METHOD INTERNAL GetNumberOfAssertsForTest : UINT
VAR_INPUT
    CompleteTestInstancePath : T_MaxString;
END_VAR
VAR
    Counter : UINT;
    NumberOfAsserts : UINT := 0;
END_VAR
IF TotalAsserts > 0 THEN
    FOR Counter := 1 TO TotalAsserts BY 1 DO
        IF AssertResults[Counter].TestInstancePath = CompleteTestInstancePath THEN
            NumberOfAsserts := NumberOfAsserts + 1;
        END_IF
    END_FOR
END_IF

GetNumberOfAssertsForTest := NumberOfAsserts;
END_METHOD

(*
    This method is called in every assert and returns whether this particular assert has already been called.
    The reason one would like to know whether this assert has already been reported or not is to not report it several
    times to any logging service. Because a test-suite can consist of several tests, and certain tests can require the
    test to run over several cycles it means that certain asserts could be called several times and thus we need to
    keep track of which asserts we've already reported. The user of the framework should not need to care for any of
    this and he/she should be able to call the asserts in any way they find suitable.

    To know what assert this is we need to check for the total combination of:
    - Test message
    - Test instance path
    - Expected value
    - Actual value
    Theoretically we can have a situation where a test has three different asserts, each and one with the same test
    message/test instance path/actual value/expected value but called within the same or different cycles. In order for
    us to handle all situations we need a simple algorithm that works according to:
    - Keep track of how many instances the combination of test message/test instance path/expected value/actual value
      we have. So for example, if we have called Assert(Exp := 5, Act := 5, 'Hello there', 'PRG.InstanceTestSuite.Test')
      two times in one cycle, we have two instances of that combination. This is done according to:
    - Iterate all existing reports.
      - If we have a new PLC-cycle, set the current detection-count to zero.
      - If new report does not match in any of the above fields, create it (together with current PLC-cycle).
        Also store the information that we have one instance of this combination and +1 on the detection-count.
      - If new report matches in all of the above, +1 in the detection-count. If this detection-count is larger than
        the stored detection-count for this combination, create a new report and add +1 to the storage of
        the detection-count.
*)
METHOD INTERNAL ReportResult
VAR_INPUT
    ExpectedSize : UDINT;
    ExpectedTypeClass : IBaseLibrary.TypeClass;
    ExpectedValue : POINTER TO BYTE;
    ActualSize : UDINT;
    ActualTypeClass : IBaseLibrary.TypeClass;
    ActualValue : POINTER TO BYTE;
    Message : T_MaxString;
    TestInstancePath : T_MaxString;
END_VAR
VAR_OUTPUT
    AlreadyReported : BOOL := FALSE;
END_VAR
VAR
    LocationIndex : UINT;
    DataTypesNotEquals : BOOL;
    DataSizeNotEquals : BOOL;
    DataContentNotEquals : BOOL;
    CurrentCycleCount : UDINT;
    IteratorCounter : UINT;
    DetectionCountTemp : UINT := 0;
    FoundOne : BOOL;
    AdditionalIdenticalAssert : BOOL;
END_VAR
IF NOT FirstCycleExecuted THEN
    GetCurrentTaskIndex();
    FirstCycleExecuted := TRUE;
END_IF

CurrentCycleCount := TwinCAT_SystemInfoVarList._TaskInfo[GetCurrentTaskIndex.index].CycleCount;
(* Is current cycle the same as the last call to this method?
   If not, reset the detection count *)
IF CurrentCycleCount <> CycleCount THEN
    CopyDetectionCountAndResetDetectionCountInThisCycle();
END_IF

FOR IteratorCounter := 1 TO TotalAsserts BY 1 DO
      IF F_IsAnyEqualToUnionValue(ExpectedOrActual := AssertResultInstances[IteratorCounter].AssertResult.Expected,
                                  ExpectedOrActualSize := ExpectedSize,
                                  ExpectedOrActualTypeClass := ExpectedTypeClass,
                                  ExpectedOrActualValue := ExpectedValue) AND
         F_IsAnyEqualToUnionValue(ExpectedOrActual := AssertResultInstances[IteratorCounter].AssertResult.Actual,
                                  ExpectedOrActualSize := ActualSize,
                                  ExpectedOrActualTypeClass := ActualTypeClass,
                                  ExpectedOrActualValue := ActualValue) AND
        AssertResultInstances[IteratorCounter].AssertResult.Message = Message AND
        AssertResultInstances[IteratorCounter].AssertResult.TestInstancePath = TestInstancePath THEN
            AssertResultInstances[IteratorCounter].DetectionCountThisCycle :=
                AssertResultInstances[IteratorCounter].DetectionCountThisCycle + 1;
            FoundOne := TRUE;
        IF AssertResultInstances[IteratorCounter].DetectionCountThisCycle >
            AssertResultInstances[IteratorCounter].DetectionCount THEN // This assert is new
            AdditionalIdenticalAssert := TRUE;
        END_IF
        EXIT;
    END_IF
END_FOR

// If not found anything, create the first
IF NOT FoundOne THEN
    // No existing match found, create a new entry
    AddAssertResult(ExpectedSize := ExpectedSize,
                    ExpectedTypeClass := ExpectedTypeClass,
                    ExpectedValue := ExpectedValue,
                    ActualSize := ActualSize,
                    ActualTypeClass := ActualTypeClass,
                    ActualValue := ActualValue,
                    Message := Message, TestInstancePath := TestInstancePath);

    CreateAssertResultInstance(ExpectedSize := ExpectedSize,
                               ExpectedTypeClass := ExpectedTypeClass,
                               ExpectedValue := ExpectedValue,
                               ActualSize := ActualSize,
                               ActualTypeClass := ActualTypeClass,
                               ActualValue := ActualValue,
                               Message := Message, TestInstancePath := TestInstancePath);
// An additional instance of this assert needs to be created
ELSIF AdditionalIdenticalAssert THEN
    AddAssertResult(ExpectedSize := ExpectedSize,
                    ExpectedTypeClass := ExpectedTypeClass,
                    ExpectedValue := ExpectedValue,
                    ActualSize := ActualSize,
                    ActualTypeClass := ActualTypeClass,
                    ActualValue := ActualValue,
                    Message := Message, TestInstancePath := TestInstancePath);
// In all other cases, this assert has already been reported, we don't need to do anything
ELSE
    AlreadyReported := TRUE;
END_IF

// Update the cycle count
CycleCount := TwinCAT_SystemInfoVarList._TaskInfo[GetCurrentTaskIndex.index].CycleCount;
END_METHOD

END_FUNCTION_BLOCK

// POUs/FB_FileControl
// This functionblock can open, close, read, write and delete files on the local filesystem
FUNCTION_BLOCK FB_FileControl
VAR
    FileAccessMode : SysFile.ACCESS_MODE := SysFile.AM_APPEND_PLUS; // Append_Plus creates the file if it doesn't exist yet. 
    FileHandle : SysFile.SysTypes.RTS_IEC_HANDLE;
END_VAR

// Closes the currently opened file.
METHOD PUBLIC Close : SysFile.SysTypes.RTS_IEC_RESULT;
IF FileHandle <> SysFile.SysTypes.RTS_INVALID_HANDLE THEN
    Close := SysFile.SysFileClose(hFile := FileHandle);
ELSE
    Close := SysDir.CmpErrors.Errors.ERR_INVALID_HANDLE;
END_IF
END_METHOD

// Deletes a file specified by name, if it exists.
METHOD PUBLIC Delete : SysFile.SysTypes.RTS_IEC_RESULT;
VAR_INPUT
    // File name can contain an absolute or relative path to the file. Path entries must be separated with a forward slash (/)
    FileName : T_MaxString;
END_VAR
Delete := SysFile.SysFileDelete(szFileName := FileName);
END_METHOD

// Opens a file
METHOD PUBLIC Open : SysFile.SysTypes.RTS_IEC_RESULT;
VAR_INPUT
    FileName : T_MaxString := 'filepath/output.xml';  // File name can contain an absolute or relative path to the file. Path entries must be separated with a Slash (/)
    FileAccessMode : SysFile.ACCESS_MODE := SysFile.ACCESS_MODE.AM_APPEND_PLUS;
END_VAR
FileHandle := SysFile.SysFileOpen(szFile := Filename,
                                  am := FileAccessMode,
                                  pResult := ADR(Open));
END_METHOD

// Reads a file from disk into the buffer
METHOD PUBLIC Read : SysFile.SysTypes.RTS_IEC_RESULT;
VAR_INPUT
    BufferPointer : POINTER TO BYTE; // Call with ADR();
    Size : UDINT; // Call with SIZEOF(); 
END_VAR
VAR_OUTPUT
    FileSize : SysFile.SysTypes.RTS_IEC_SIZE;
END_VAR
IF FileHandle <> SysFile.SysTypes.RTS_INVALID_HANDLE THEN
    FileSize := SysFile.SysFileRead(hFile := FileHandle, 
                                    pbyBuffer := BufferPointer,
                                    ulSize := Size,
                                    pResult := ADR(Read));
ELSE
    Read := SysDir.CmpErrors.Errors.ERR_INVALID_HANDLE;
END_IF
END_METHOD

// Writes the contents of the buffer into a file.
METHOD PUBLIC Write : SysFile.SysTypes.RTS_IEC_RESULT;
VAR_INPUT
    BufferPointer : POINTER TO BYTE; // Call with ADR();
    Size : UDINT; // Call with SIZEOF();
END_VAR
IF FileHandle <> SysFile.SysTypes.RTS_INVALID_HANDLE THEN
    SysFile.SysFileWrite(hFile := FileHandle,
                         pbyBuffer := BufferPointer,
                         ulSize := Size,
                         pResult := ADR(Write));
ELSE
    Write := SysDir.CmpErrors.Errors.ERR_INVALID_HANDLE;
END_IF
END_METHOD

END_FUNCTION_BLOCK

// POUs/FB_StreamBuffer
// This functionblock acts as a stream buffer for use with FB_XmlControl
FUNCTION_BLOCK FB_StreamBuffer 
VAR
    _PointerToStringBuffer : POINTER TO BYTE;
    _BufferSize : UDINT;
    _Length : UDINT;
END_VAR

// Appends a string to the buffer
PROPERTY Append : T_MaxString
SET
VAR
    ByteIn : POINTER TO BYTE;
    ByteBuffer : POINTER TO BYTE;
END_VAR
ByteIn := ADR(Append); 
ByteBuffer := _PointerToStringBuffer + _Length; // set start address

WHILE ByteIn^ <> 0 AND (_Length < _BufferSize ) DO
    ByteBuffer^ := ByteIn^; //Copy the 1st byte
    _Length := _Length + 1; // set new buffer length
    ByteIn := ByteIn + 1; // calculate new start address 
    ByteBuffer := ByteBuffer + 1; // calculate new start address 
END_WHILE;

ByteBuffer := _PointerToStringBuffer + _Length; // String End
ByteBuffer^ := 0; // null terminated string
END_SET
END_PROPERTY

// Read current Buffersize
PROPERTY BufferSize : UDINT
GET
BufferSize := _BufferSize;
END_GET
END_PROPERTY

// Clears the buffer and sets the length to 0
METHOD PUBLIC Clear
VAR
	Count : UDINT;
END_VAR
IF (_PointerToStringBuffer = 0) OR (_BufferSize = 0) THEN
    RETURN;
END_IF

FOR Count := 0 TO (_BufferSize - 1) DO
    _PointerToStringBuffer[Count] := 0;
END_FOR

_Length := 0;
END_METHOD

// Copies a string from the character buffer
METHOD PUBLIC Copy : T_MaxString
VAR_INPUT
    StartPos : UDINT;
    EndPos : UDINT;
END_VAR
VAR_OUTPUT
    CopyLen : UDINT;
    XmlError : E_XmlError;
END_VAR
VAR
    Loop : UDINT;
    PointerToByteToCopy : POINTER TO BYTE;
    PointerToBuffer : POINTER TO BYTE;
    CurPos : UDINT;
END_VAR
Loop := 0;
PointerToByteToCopy := ADR(Copy);
PointerToBuffer := _PointerToStringBuffer + StartPos - 1;

WHILE(Loop < SIZEOF(Copy)) AND (StartPos - 1 + Loop < _Length) AND (StartPos + Loop < EndPos) DO
    PointerToByteToCopy^ := PointerToBuffer^;
    Loop := Loop + 1;
    PointerToByteToCopy := ADR(Copy) + Loop;
    PointerToBuffer := _PointerToStringBuffer + StartPos + Loop -1;
END_WHILE;

IF Loop = SIZEOF(Copy) THEN
    XmlError := E_XmlError.ErrorStringLen;
ELSIF StartPos - 1 + Loop = _Length THEN
    XmlError := E_XmlError.ErrorMaxBufferLen;
ELSE
    XmlError := E_XmlError.OK;
END_IF;

PointerToByteToCopy^ := 0;
CopyLen :=  Loop;
END_METHOD

METHOD PUBLIC CutOff : T_MaxString
VAR_INPUT
    StartPos : UDINT;
END_VAR
VAR_OUTPUT
    CutLen : UDINT; 
    XmlError : E_XmlError;
END_VAR
VAR
    Loop : UDINT;
    PointerToByteToCut : POINTER TO BYTE;
    PointerToByteBuffer : POINTER TO BYTE;
END_VAR
Loop := 0;
PointerToByteToCut := ADR(CutOff);
PointerToByteBuffer := _PointerToStringBuffer + StartPos - 1;

WHILE PointerToByteBuffer^ <> 0 AND(Loop < SIZEOF(CutOff)) AND StartPos -1  + Loop < _Length DO
    PointerToByteToCut^ := PointerToByteBuffer^;
    Loop := Loop + 1;
    PointerToByteToCut := ADR(CutOff) + Loop;
    PointerToByteBuffer := _PointerToStringBuffer + StartPos - 1 + Loop;
END_WHILE;

IF PointerToByteBuffer^ = 0 THEN
    XmlError := E_XmlError.OK;
ELSIF Loop = SIZEOF(CutOff) THEN
    XmlError := E_XmlError.ErrorStringLen;
ELSIF StartPos - 1 + Loop = _Length THEN
    XmlError := E_XmlError.ErrorMaxBufferLen;
END_IF;

PointerToByteToCut^ := 0;
_Length := StartPos -1;

PointerToByteBuffer := _PointerToStringBuffer + StartPos - 1;
PointerToByteBuffer^ := 0;

CutLen := Loop;
END_METHOD

(* 
    Find a searchstring in the buffer and returns its position.
    It's possible to add a preffered startposition within buffer
*)
METHOD PUBLIC Find : UDINT
VAR_INPUT
    SearchString : STRING;
    StartPos : UDINT;
END_VAR
VAR
    Loop : UDINT;
    Search : UDINT;
    PointerToBuffer : POINTER TO BYTE;
    PointerToSearch : POINTER TO BYTE;
END_VAR
Loop := 0;
Search := 0;

PointerToBuffer := _PointerToStringBuffer + StartPos;
PointerToSearch := ADR(SearchString);

WHILE(PointerToSearch^ <> 0 ) AND Loop + StartPos < _Length DO
    IF PointerToBuffer^ <> PointerToSearch^ THEN
        Loop := Loop + 1;
        PointerToBuffer := _PointerToStringBuffer + StartPos + Loop;
        PointerToSearch := ADR(SearchString);
        Search := 0;
    ELSE
        Search := Search + 1;
        PointerToBuffer := _PointerToStringBuffer + StartPos + Loop + Search;
        PointerToSearch := ADR(SearchString ) + Search;
    END_IF;
END_WHILE;
Find := Loop + 1 + StartPos;
END_METHOD

METHOD PUBLIC FindBack : UDINT
VAR_INPUT
    SearchString : T_MaxString;
END_VAR
VAR
    Loop : UDINT;
    Search : UDINT;
    PointerToBuffer : POINTER TO BYTE;
    PointerToSearch : POINTER TO BYTE;
END_VAR
Loop := 0;
Search := 0;

PointerToBuffer := _PointerToStringBuffer + _Length;
PointerToSearch := ADR(SearchString);

WHILE(PointerToSearch^ <> 0) AND Loop < _Length DO
    IF PointerToBuffer^ <> PointerToSearch^ THEN
        Loop := Loop + 1;
        PointerToBuffer := _PointerToStringBuffer + _Length - Loop;
        PointerToSearch := ADR(SearchString);
        Search := 0;
    ELSE
        Search := Search + 1;
        PointerToBuffer := _PointerToStringBuffer + _Length - Loop + Search;
        PointerToSearch := ADR(SearchString ) + Search;
    END_IF;
END_WHILE;
FindBack := _Length - Loop + 1;
END_METHOD

// Gets/Sets the current length (in bytes) of the streambuffer
PROPERTY Length : UDINT
GET
Length := _Length;
END_GET
SET
_Length := Length;
END_SET
END_PROPERTY

METHOD PUBLIC SetBuffer : BOOL;
VAR_INPUT
    PointerToBufferAddress : POINTER TO BYTE; // Set buffer address (ADR ...)
    SizeOfBuffer : UDINT; // Set buffer size (SIZEOF ...)
END_VAR
IF (PointerToBufferAddress = 0) OR (SizeOfBuffer = 0) THEN
    SetBuffer := FALSE;
    RETURN;
END_IF;

_BufferSize := SizeOfBuffer;
_PointerToStringBuffer := PointerToBufferAddress;

SetBuffer := TRUE;
END_METHOD

END_FUNCTION_BLOCK

// POUs/FB_XmlControl
(*
    Organizes parsing and composing of XML data. Data can be treated as STRING or char array.
    Buffer size of file can be set via GVL_Param_TcUnit (xUnitBufferSize)
*)
FUNCTION_BLOCK FB_XmlControl
VAR
    XmlBuffer : FB_StreamBuffer;
    TagListBuffer : FB_StreamBuffer;
    Tags : T_MaxString;
    TagListSeekBuffer : FB_StreamBuffer;
    TagsSeek : STRING;
    TagBuffer : FB_StreamBuffer;
    Tag : T_MaxString;
    TagOpen: BOOL;
    Select : UDINT;
    SearchPosition : UDINT; 
END_VAR
VAR CONSTANT
    TAG_OPEN : STRING(1) := '<';
    TAG_CLOSE : STRING(1) := '>';
    END_TAG_CLOSE : STRING(2) := '/>';
    SPACE : STRING(1) := ' ';
    EQUALS : STRING(1) := '=';
    QUOTE : STRING(1) := '"';
    BACK_SLASH : STRING(1) := '\';
    FORWARD_SLASH : STRING(1) := '/';
    OPEN_COMMENT : STRING(5) := '<!-- ';
    CLOSE_COMMENT : STRING(4) := ' -->';
    TAB : STRING(2) := '$T';
    CR_LF : STRING(4) := '$R$N';

    // $OD : ASCII code for carriage return (CR)
    // $$ : to add a $R
    // $' : to add ' (apostrophe)
    // $L or $l : line feed
    // $N or $n : new line
    // $P or $p : next page
    // $R or $r : end of line
END_VAR

// Clears the contents of the entire buffer.
METHOD PUBLIC ClearBuffer
SearchPosition := 0;
TagListSeekBuffer.Length := 0;
XmlBuffer.Length := 0;
TagsSeek := '';
Tag := '';
END_METHOD

(*
    Closes a Tag:
    XML: <MyTag />'

    Method: XML.CloseTag();
*)
METHOD PUBLIC CloseTag : T_MaxString
VAR
    ClosedTag : T_MaxString;
END_VAR
IF TagOpen THEN
    XmlBuffer.Append := END_TAG_CLOSE;
    Select := TagListBuffer.FindBack(SearchString := FORWARD_SLASH);
    ClosedTag := TagListBuffer.CutOff(StartPos := Select);
    TagOpen := FALSE;
ELSE
    Select := TagListBuffer.FindBack(SearchString := FORWARD_SLASH);
    ClosedTag := TagListBuffer.CutOff(StartPos := Select);
    XmlBuffer.Append := TAG_OPEN;
    XmlBuffer.Append := ClosedTag;
    XmlBuffer.Append := TAG_CLOSE;
END_IF

CloseTag := ClosedTag;
END_METHOD

PROPERTY Length : UDINT
GET
Length := XmlBuffer.Length;
END_GET
END_PROPERTY

(*
    Adds a comment
    XML: <!-- MyComment -->

    XML.NewComment(Comment: = 'MyComment');
*)
METHOD PUBLIC NewComment
VAR_INPUT
    Comment : T_MaxString;
END_VAR
IF TagOpen THEN
    XmlBuffer.Append := TAG_CLOSE;
    TagOpen := FALSE;
END_IF;
XmlBuffer.Append := OPEN_COMMENT;
XmlBuffer.Append := Comment;
XmlBuffer.Append := CLOSE_COMMENT;
END_METHOD

(*
    Must be called after opening a new tag

    XML.NewParameter(Name: = 'ParaName', Value: = 'Value');
*)
METHOD PUBLIC NewParameter
VAR_INPUT
    Name : T_MaxString;
    Value : T_MaxString;
END_VAR
XmlBuffer.Append := SPACE;
XmlBuffer.Append := Name;
XmlBuffer.Append := EQUALS;
XmlBuffer.Append := QUOTE;
XmlBuffer.Append := Value;
XmlBuffer.Append := QUOTE;
END_METHOD

(*
    Creates a new Tag:
    XML: <MyTag>

    XML.NewTag(Name: = 'MyTag');
*)
METHOD PUBLIC NewTag
VAR_INPUT
    Name : T_MaxString;
END_VAR
IF TagOpen THEN
    XmlBuffer.Append := TAG_CLOSE;
END_IF;
XmlBuffer.Append := TAG_OPEN;
XmlBuffer.Append := Name;
TagOpen := TRUE;
TagListBuffer.Append := FORWARD_SLASH;
TagListBuffer.Append := Name;
END_METHOD

METHOD PUBLIC NewTagData
VAR_INPUT
    Data : T_MaxString;
END_VAR
XmlBuffer.Append := TAG_CLOSE;
XmlBuffer.Append := Data;
TagOpen := FALSE;
END_METHOD

METHOD PUBLIC SetBuffer
VAR_INPUT
    PointerToBuffer : POINTER TO BYTE; // ADR(..)
    SizeOfBuffer : UDINT; // SIZEOF(..)
END_VAR
XmlBuffer.SetBuffer(PointerToBufferAddress:= PointerToBuffer, SizeOfBuffer := SizeOfBuffer);
TagListBuffer.SetBuffer(PointerToBufferAddress := ADR(Tags), SizeOfBuffer := SIZEOF(Tags));
TagListSeekBuffer.SetBuffer(PointerToBufferAddress := ADR(TagsSeek), SizeOfBuffer := SIZEOF(TagsSeek));
TagBuffer.SetBuffer(PointerToBufferAddress := ADR(Tag), SizeOfBuffer := SIZEOF(Tag));
END_METHOD

(*
    Jump to the beginning of the XML data
    XML.ToStartBuffer();
*)
METHOD PUBLIC ToStartBuffer
SearchPosition := 0;
TagListSeekBuffer.Length := 0;
TagsSeek := '';
Tag := '';
END_METHOD

(*
    Add your own preffered fileheader like:
    XML: <?xml version="1.0" encoding="UTF-8"?>
    
    Start with calling this method before appending any other tags!

    XML.WriteDocumentHeader('<?xml version="1.0" encoding="UTF-8"?>');
*)
METHOD PUBLIC WriteDocumentHeader
VAR_INPUT
    Header : T_MaxString;
END_VAR
XmlBuffer.Append := Header;
END_METHOD

END_FUNCTION_BLOCK

// POUs/FB_TcUnitRunner
// This function block is responsible for holding track of the tests and executing them.
FUNCTION_BLOCK FB_TcUnitRunner
VAR
    // Indication of whether all test suites have reported that they are finished
    AllTestSuitesFinished : BOOL := FALSE;
    AllTestSuitesFinishedTrigger : R_TRIG;

    //Test result information
    TestResults : FB_TestResults;

    (* Prints the results to ADS so that Visual Studio can display the results.
       This test result formatter can be replaced with something else than ADS *)
    AdsTestResultLogger : FB_AdsTestResultLogger(TestResults);
    TestResultLogger : I_TestResultLogger := AdsTestResultLogger;

    (* If this flag is set, it means that some external event triggered the
       request to abort running the test suites *)
    AbortRunningTestSuites : BOOL;

    // Publishes a xUnit compatible XML file
    xUnitXmlPublisher : FB_xUnitXmlPublisher(TestResults);
    XmlTestResultPublisher : I_TestResultLogger := xUnitXmlPublisher;
END_VAR

(* This function sets a flag which makes the runner stop running the tests
   in the test suites *)
METHOD INTERNAL AbortRunningTestSuiteTests
AbortRunningTestSuites := TRUE;
END_METHOD

// This runs all the test suites in parallel
METHOD INTERNAL RunTestSuiteTests
VAR
    Counter : UINT := 0;
    BusyPrinting : BOOL;
    (* We need to hold a temporary state of the statistics 
       as we don't consider the tests to be completely finished until all test suites have executed completely.
       The reason we want to do it this way is because a test suite can run over several cycles. Only once all tests
       are finished (which might take many cycles), do we gather correct statistics *)
    NumberOfTestSuitesFinished : UINT := 0;
END_VAR
IF GVL_TcUnit.StartedAt = 0 THEN
    GVL_TcUnit.StartedAt := F_GetCpuCounterAs64bit(GVL_TcUnit.GetCpuCounter);
END_IF

// Run TcUnit test suites
IF NOT AllTestSuitesFinished THEN
    IF GVL_TcUnit.NumberOfInitializedTestSuites = 0 THEN
        AllTestSuitesFinished := TRUE;
    ELSIF GVL_TcUnit.NumberOfInitializedTestSuites > 0 THEN
        FOR Counter := 1 TO GVL_TcUnit.NumberOfInitializedTestSuites BY 1 DO
            IF GVL_TcUnit.TestSuiteAddresses[Counter]^.AreAllTestsFinished() THEN
                NumberOfTestSuitesFinished := NumberOfTestSuitesFinished + 1;
            ELSE
                GVL_TcUnit.CurrentTestSuiteBeingCalled := GVL_TcUnit.TestSuiteAddresses[Counter];
				GVL_TcUnit.CurrentTestSuiteBeingCalled^.SetStartedAtIfNotSet(Timestamp := F_GetCpuCounterAs64bit(GVL_TcUnit.GetCpuCounter));
                GVL_TcUnit.CurrentTestSuiteBeingCalled^();
				// This is not an efficient way to set the duration
				IF GVL_TcUnit.TestSuiteAddresses[Counter]^.AreAllTestsFinished() THEN
					GVL_TcUnit.CurrentTestSuiteBeingCalled^.CalculateDuration(FinishedAt := F_GetCpuCounterAs64bit(GVL_TcUnit.GetCpuCounter));
				END_IF
            END_IF
        END_FOR
        (* Check if some event triggered an abortion of running the tests, in that case abort it now.
           This can be accomplished by setting the result of the test suites run to finished. *)
        IF AbortRunningTestSuites THEN
            NumberOfTestSuitesFinished := GVL_TcUnit.NumberOfInitializedTestSuites;
        END_IF

        IF NumberOfTestSuitesFinished = GVL_TcUnit.NumberOfInitializedTestSuites THEN
            AllTestSuitesFinished := TRUE;
        END_IF
    END_IF
END_IF

// Store test suite results continuously
TestResults();

// Log test suite results continuously
TestResultLogger.LogTestSuiteResults();

// Publish the xUnit Xml file once if enabled
XmlTestResultPublisher.LogTestSuiteResults();

// Run the buffered ADS logger
GVL_TcUnit.AdsMessageQueue();
END_METHOD

// This runs all the test suites in sequence (one after the other)
METHOD INTERNAL RunTestSuiteTestsInSequence
VAR_INPUT
    TimeBetweenTestSuitesExecution : TIME; // Time delay between a test suite is finished and the next test suite starts
END_VAR
VAR
    BusyPrinting : BOOL;
    (* We need to hold a temporary state of the statistics
       as we don't consider the tests to be completely finished until all test suites have executed completely.
       The reason we want to do it this way is because a test suite can run over several cycles. Only once all tests
       are finished (which might take many cycles), do we gather correct statistics *)
    NumberOfTestSuitesFinished : UINT := 0;
END_VAR
VAR_INST
    (* This variable holds which current test suite is being called, as we are running
       each one in a sequence (one by one) *)
     CurrentlyRunningTestSuite : UINT := 1;
     TimerBetweenExecutionOfTestSuites : TOF;
END_VAR
IF GVL_TcUnit.StartedAt = 0 THEN
    GVL_TcUnit.StartedAt := F_GetCpuCounterAs64bit(GVL_TcUnit.GetCpuCounter);
END_IF

TimerBetweenExecutionOfTestSuites(PT := TimeBetweenTestSuitesExecution);
// Run TcUnit test suites
IF NOT AllTestSuitesFinished THEN
    IF GVL_TcUnit.NumberOfInitializedTestSuites = 0 THEN
        AllTestSuitesFinished := TRUE;
    ELSIF GVL_TcUnit.NumberOfInitializedTestSuites > 0 THEN
        IF TimerBetweenExecutionOfTestSuites.Q THEN
            TimerBetweenExecutionOfTestSuites.IN := FALSE;
        END_IF
        IF GVL_TcUnit.TestSuiteAddresses[CurrentlyRunningTestSuite]^.AreAllTestsFinished() THEN
            IF CurrentlyRunningTestSuite <> GVL_TcUnit.NumberOfInitializedTestSuites THEN
                NumberOfTestSuitesFinished := NumberOfTestSuitesFinished + 1;
                CurrentlyRunningTestSuite := CurrentlyRunningTestSuite + 1;
                TimerBetweenExecutionOfTestSuites.IN := TRUE;
				GVL_TcUnit.CurrentTestSuiteBeingCalled^.CalculateDuration(FinishedAt := F_GetCpuCounterAs64bit(GVL_TcUnit.GetCpuCounter));
            END_IF
        ELSIF NOT TimerBetweenExecutionOfTestSuites.Q THEN
            GVL_TcUnit.CurrentTestSuiteBeingCalled := GVL_TcUnit.TestSuiteAddresses[CurrentlyRunningTestSuite];
			GVL_TcUnit.CurrentTestSuiteBeingCalled^.SetStartedAtIfNotSet(Timestamp := F_GetCpuCounterAs64bit(GVL_TcUnit.GetCpuCounter));
            GVL_TcUnit.CurrentTestSuiteBeingCalled^();
			// This is not an efficient way to set the duration
			IF GVL_TcUnit.TestSuiteAddresses[CurrentlyRunningTestSuite]^.AreAllTestsFinished() THEN
				GVL_TcUnit.CurrentTestSuiteBeingCalled^.CalculateDuration(FinishedAt := F_GetCpuCounterAs64bit(GVL_TcUnit.GetCpuCounter));
			END_IF
        END_IF
        (* Check if some event triggered an abortion of running the tests, in that case abort it now.
           This can be accomplished by setting the result of the test suites run to finished. *)
        IF AbortRunningTestSuites THEN
            NumberOfTestSuitesFinished := GVL_TcUnit.NumberOfInitializedTestSuites;
        END_IF
        IF NumberOfTestSuitesFinished = GVL_TcUnit.NumberOfInitializedTestSuites THEN
            AllTestSuitesFinished := TRUE;
        END_IF
    END_IF
END_IF

// Store test suite results continuously
TestResults();

// Log test suite results continuously
TestResultLogger.LogTestSuiteResults();

// Publish the xUnit Xml file once if enabled
XmlTestResultPublisher.LogTestSuiteResults();

// Run the buffered ADS logger
GVL_TcUnit.AdsMessageQueue();
END_METHOD

END_FUNCTION_BLOCK

// POUs/FB_TestResults
// This function block holds results of the complete test run, i.e. results for all test suites
FUNCTION_BLOCK FB_TestResults IMPLEMENTS I_TestResults
VAR
    // Test results
    TestSuiteResults : ST_TestSuiteResults;

    // Misc variables
    StoringTestSuiteResultNumber : UINT(1..GVL_Param_TcUnit.MaxNumberOfTestSuites);
    StoringTestSuiteTrigger : R_TRIG;
    StoredTestSuiteResults : BOOL;
    StoredGeneralTestResults : BOOL;
    NumberOfTestsToAnalyse : UINT(1..GVL_Param_TcUnit.MaxNumberOfTestsForEachTestSuite);
END_VAR
VAR_TEMP
    TestSuiteName : T_MaxString;
    TestName : T_MaxString;

    TestsInTestSuiteCounter : UINT(1..GVL_Param_TcUnit.MaxNumberOfTestsForEachTestSuite);

    TestToBeStored : FB_Test;
    GeneralTestResultsTestSuitesCounter : UINT(1..GVL_Param_TcUnit.MaxNumberOfTestSuites);
END_VAR

// The body of the function block stores the test results
IF StoringTestSuiteResultNumber <= GVL_TcUnit.NumberOfInitializedTestSuites AND NOT StoredTestSuiteResults THEN
	StoringTestSuiteTrigger(CLK := GVL_TcUnit.TestSuiteAddresses[StoringTestSuiteResultNumber]^.AreAllTestsFinished());

    IF StoringTestSuiteTrigger.Q THEN
        // Remove everything except the program name + "." + test suite name
        TestSuiteName := F_RemoveInstancePathAndProjectNameFromTestInstancePath(TestInstancePath := GVL_TcUnit.TestSuiteAddresses[StoringTestSuiteResultNumber]^.GetInstancePath());

        // Store test suite name and ID
        TestSuiteResults.TestSuiteResults[StoringTestSuiteResultNumber].Name := TestSuiteName;
        TestSuiteResults.TestSuiteResults[StoringTestSuiteResultNumber].Identity := StoringTestSuiteResultNumber - 1;

        // Store number of tests in test suite
        TestSuiteResults.TestSuiteResults[StoringTestSuiteResultNumber].NumberOfTests :=
            GVL_TcUnit.TestSuiteAddresses[StoringTestSuiteResultNumber]^.GetNumberOfTests();

        // Store number of failed tests in test suite
        TestSuiteResults.TestSuiteResults[StoringTestSuiteResultNumber].NumberOfFailedTests :=
            GVL_TcUnit.TestSuiteAddresses[StoringTestSuiteResultNumber]^.GetNumberOfFailedTests();

        // Store the duration
        TestSuiteResults.TestSuiteResults[StoringTestSuiteResultNumber].Duration :=
            GVL_TcUnit.TestSuiteAddresses[StoringTestSuiteResultNumber]^.GetDuration();

        // Limit the test analyse to the max array limit of 'Tests[]' in FB_TestSuite
        NumberOfTestsToAnalyse := GVL_TcUnit.TestSuiteAddresses[StoringTestSuiteResultNumber]^.GetNumberOfTestsToAnalyse();

        // Iterate and print all tests in test suite
        FOR TestsInTestSuiteCounter := 1 TO NumberOfTestsToAnalyse BY 1 DO
            TestToBeStored := GVL_TcUnit.TestSuiteAddresses[StoringTestSuiteResultNumber]^.GetTestByPosition(TestsInTestSuiteCounter);
            // Store test name
            TestSuiteResults.TestSuiteResults[StoringTestSuiteResultNumber].TestCaseResults[TestsInTestSuiteCounter].TestName := TestToBeStored.GetName();

            // Store test class name
            TestSuiteResults.TestSuiteResults[StoringTestSuiteResultNumber].TestCaseResults[TestsInTestSuiteCounter].TestClassName :=
                F_RemoveInstancePathAndProjectNameFromTestInstancePath(GVL_TcUnit.TestSuiteAddresses[StoringTestSuiteResultNumber]^.GetInstancePath());

            // Store whether the test has failed
            TestSuiteResults.TestSuiteResults[StoringTestSuiteResultNumber].TestCaseResults[TestsInTestSuiteCounter].TestIsFailed :=
                TestToBeStored.IsFailed();

            // Store whether the test was skipped
            TestSuiteResults.TestSuiteResults[StoringTestSuiteResultNumber].TestCaseResults[TestsInTestSuiteCounter].TestIsSkipped :=
                TestToBeStored.IsSkipped();

            // Store the (first failed) assertion message
            TestSuiteResults.TestSuiteResults[StoringTestSuiteResultNumber].TestCaseResults[TestsInTestSuiteCounter].FailureMessage :=
                TestToBeStored.GetAssertionMessage();

            // Store the (first failed) assertion type
            TestSuiteResults.TestSuiteResults[StoringTestSuiteResultNumber].TestCaseResults[TestsInTestSuiteCounter].FailureType :=
                TestToBeStored.GetAssertionType();

            // Store number of assertions made
            TestSuiteResults.TestSuiteResults[StoringTestSuiteResultNumber].TestCaseResults[TestsInTestSuiteCounter].NumberOfAsserts :=
                TestToBeStored.GetNumberOfAssertions();

            // Store the duration of the test
            TestSuiteResults.TestSuiteResults[StoringTestSuiteResultNumber].TestCaseResults[TestsInTestSuiteCounter].Duration :=
                TestToBeStored.GetDuration();
        END_FOR

        IF StoringTestSuiteResultNumber = GVL_TcUnit.NumberOfInitializedTestSuites THEN
            StoredTestSuiteResults := TRUE;
        ELSE
            StoringTestSuiteResultNumber := StoringTestSuiteResultNumber + 1;
        END_IF
        StoringTestSuiteTrigger(CLK := FALSE); // Reset trigger
    END_IF
END_IF

(* If all test suites have finished running, store the general test results.
   Take care OF the special CASE where no tests have NOT yet been defined *)
IF GVL_TcUnit.NumberOfInitializedTestSuites = 0 AND (NOT StoredGeneralTestResults) THEN
    StoredGeneralTestResults := TRUE;
    StoredTestSuiteResults := TRUE;
ELSIF StoringTestSuiteResultNumber = GVL_TcUnit.NumberOfInitializedTestSuites AND_THEN
    GVL_TcUnit.TestSuiteAddresses[StoringTestSuiteResultNumber]^.AreAllTestsFinished() AND StoredTestSuiteResults AND (NOT StoredGeneralTestResults) THEN
    TestSuiteResults.NumberOfTestSuites := GVL_TcUnit.NumberOfInitializedTestSuites;
	GVL_TcUnit.Duration := LWORD_TO_LREAL(F_GetCpuCounterAs64bit(GVL_TcUnit.GetCpuCounter) - GVL_TcUnit.StartedAt) * GVL_TcUnit.HundredNanosecondToSecond; // Seconds
    TestSuiteResults.Duration := GVL_TcUnit.Duration;
    FOR GeneralTestResultsTestSuitesCounter := 1 TO GVL_TcUnit.NumberOfInitializedTestSuites BY 1 DO
        TestSuiteResults.NumberOfTestCases := TestSuiteResults.NumberOfTestCases + TestSuiteResults.TestSuiteResults[GeneralTestResultsTestSuitesCounter].NumberOfTests;
        TestSuiteResults.NumberOfSuccessfulTestCases := TestSuiteResults.NumberOfSuccessfulTestCases +
                                                        (TestSuiteResults.TestSuiteResults[GeneralTestResultsTestSuitesCounter].NumberOfTests -
                                                         TestSuiteResults.TestSuiteResults[GeneralTestResultsTestSuitesCounter].NumberOfFailedTests);
        TestSuiteResults.NumberOfFailedTestCases := TestSuiteResults.NumberOfFailedTestCases + TestSuiteResults.TestSuiteResults[GeneralTestResultsTestSuitesCounter].NumberOfFailedTests;
    END_FOR
    StoredGeneralTestResults := TRUE;
END_IF

// Returns whether the storing of the test results is finished
METHOD PUBLIC GetAreTestResultsAvailable : BOOL
GetAreTestResultsAvailable := (StoredTestSuiteResults AND StoredGeneralTestResults);
END_METHOD

METHOD PUBLIC GetTestSuiteResults : REFERENCE TO ST_TestSuiteResults;
GetTestSuiteResults REF=TestSuiteResults;
END_METHOD

END_FUNCTION_BLOCK

// POUs/FB_TestSuite
(* This function block is responsible for holding the internal state of the test suite.
   Every test suite can have one or more tests, and every test can do one or more asserts.
   It's also responsible for providing all the assert-methods for asserting different data types.
   Only failed assertions are recorded.
*)
{attribute 'call_after_init'}
{attribute 'reflection'}
FUNCTION_BLOCK FB_TestSuite
VAR
    {attribute 'instance-path'}
    {attribute 'noinit'}
    InstancePath : T_MaxString;

    (* We need to have access to specific information of the current task that this test suite
       is executed in. This is for instance necessary when we need to know whether a test is
       defined already. The definition of a test that is defined already is that we call on it
       with the same name twice in the same cycle *)
    GetCurrentTaskIndex : GETCURTASKINDEX;

    NumberOfTests : UINT(0..GVL_Param_TcUnit.MaxNumberOfTestsForEachTestSuite) := 0;
    Tests : ARRAY[1..GVL_Param_TcUnit.MaxNumberOfTestsForEachTestSuite] OF FB_Test;
    (* Rising trigger of whether we have already notified the user of that the test name pointed to by the current
       position is a duplicate *)
    TestDuplicateNameTrigger : ARRAY[1..GVL_Param_TcUnit.MaxNumberOfTestsForEachTestSuite] OF R_TRIG;
    (* Last cycle count index for a specific test. Used to detect whether this test has already been defined in the
       current test suite *)
    TestCycleCountIndex : ARRAY[1..GVL_Param_TcUnit.MaxNumberOfTestsForEachTestSuite] OF UDINT;

    AssertResults : FB_AssertResultStatic;
    AssertArrayResults : FB_AssertArrayResultStatic;

    (* Prints the failed asserts to ADS so that Visual Studio can display the assert message.
       This assert formatter can be replaced with something else than ADS *)
    AdsAssertMessageFormatter : FB_AdsAssertMessageFormatter;
    AssertMessageFormatter : I_AssertMessageFormatter := AdsAssertMessageFormatter;

    (* Stores the CPU cycle count with 100ns precision. It also is an indication whether this 
       test suite has started running its tests (> 0 means it has started) *)
    StartedAt : LWORD;

    (* Duration it took to run all tests in this testsuite - including the overhead from TcUnit
       in seconds *)
    Duration : LREAL;

    // Number of ordered tests (created by TEST_ORDERED()) that this test suite contains
    NumberOfOrderedTests : UINT(0..GVL_Param_TcUnit.MaxNumberOfTestsForEachTestSuite);
END_VAR

METHOD INTERNAL AddTest : REFERENCE TO FB_Test
VAR_INPUT
    TestName : T_MaxString;
    IsTestOrdered : BOOL;
END_VAR
VAR
    IteratorCounter : UINT;
    ErrorMessage : T_MaxString;
    TestInstancePath : T_MaxString;
    FunctionCallResult : DINT;
    CycleCount : UDINT;
    TestWithThisNameAlreadyExists : BOOL := FALSE;
    LowerCasedTestName : T_MaxString;
    TrimmedTestName : T_MaxString;
    IgnoreCurrentTestCase : BOOL;
    NumberOfTestsToAnalyse : UINT(1..GVL_Param_TcUnit.MaxNumberOfTestsForEachTestSuite);
END_VAR
GVL_TcUnit.IgnoreCurrentTest := FALSE; // Reset the ignore current test flag

TrimmedTestName := F_LTrim(in := TestName);
TrimmedTestName := F_RTrim(in := TrimmedTestName);
LowerCasedTestName := F_ToLCase(in := TrimmedTestName);

// If test should be disabled, make sure to remove the "disabled_"-part of it from the test name
IF FIND(STR1 := LowerCasedTestName, STR2 := 'disabled_') = 1 THEN
    IgnoreCurrentTestCase := TRUE;
    TrimmedTestName := DELETE(STR := TrimmedTestName, LEN := LEN(STR := 'disabled_'), POS := 1);
END_IF

GetCurrentTaskIndex(); // Gets the task index of where this function block instance is being run in

(* Check if the test name already exists. Make sure there are no other tests with the same name already
   added for this test suite *)

CycleCount := TwinCAT_SystemInfoVarList._TaskInfo[GetCurrentTaskIndex.index].CycleCount;

// Limit the test analyse to the max array limit of 'Tests[]'
NumberOfTestsToAnalyse := GetNumberOfTestsToAnalyse();

// Iterate all the test names that up to this point have been added for this test suite
FOR IteratorCounter := 1 TO NumberOfTestsToAnalyse BY 1 DO
    IF Tests[IteratorCounter].GetName() = TrimmedTestName THEN
        TestWithThisNameAlreadyExists := TRUE;
        // Check if a test with this name has already been called in this PLC cycle
        IF TestCycleCountIndex[IteratorCounter] = CycleCount THEN
            GVL_TcUnit.IgnoreCurrentTest := TRUE;
            (* A test with this name already exists for this test suite and has already been called in this cycle.
               Send a message notification, but only if we have not done so already. *)
            TestDuplicateNameTrigger[IteratorCounter](CLK := TRUE);
            IF TestDuplicateNameTrigger[IteratorCounter].Q THEN // Rising edge detected. We have not reported this before
                TestInstancePath := F_RemoveInstancePathAndProjectNameFromTestInstancePath(TestInstancePath :=
                                                                                           GVL_TcUnit.CurrentTestSuiteBeingCalled^.GetInstancePath());
                ErrorMessage := 'Test with name $'%s$' already exists in test suite $'';
                ErrorMessage := CONCAT(STR1 := ErrorMessage, STR2 := TestInstancePath);
                ErrorMessage := CONCAT(STR1 := ErrorMessage, STR2 := '$'');
                GVL_TcUnit.AdsMessageQueue.WriteLog(MsgCtrlMask := ADSLOG_MSGTYPE_ERROR,
                                                    MsgFmtStr := ErrorMessage,
                                                    StrArg := TrimmedTestName);
            END_IF
        END_IF
        TestCycleCountIndex[IteratorCounter] := CycleCount;
    END_IF
END_FOR

IF NOT TestWithThisNameAlreadyExists THEN
    // Test has not been found. Add it.
    Tests[IteratorCounter].SetName(Name := TrimmedTestName);
    NumberOfTests := NumberOfTests + 1;
    TestCycleCountIndex[NumberOfTests] := CycleCount;
    IF IgnoreCurrentTestCase THEN
        Tests[IteratorCounter].SetSkipped();
    END_IF

    // Extra information to be added if test is ordered (called by TEST_ORDERED())
    IF IsTestOrdered THEN
        NumberOfOrderedTests := NumberOfOrderedTests + 1;
        Tests[IteratorCounter].SetTestOrder(OrderNumber := NumberOfOrderedTests);
    END_IF
END_IF

// Check if this test should be disabled
IF IgnoreCurrentTestCase THEN
    GVL_TcUnit.IgnoreCurrentTest := TRUE;
    RETURN;
END_IF

AddTest REF= GetTestByName(TrimmedTestName);
END_METHOD

METHOD INTERNAL AddTestNameToInstancePath : T_MaxString
VAR_INPUT
    TestInstancePath : T_MaxString;
END_VAR
VAR
    CompleteTestInstancePath : T_MaxString;
END_VAR
CompleteTestInstancePath := CONCAT(STR1 := TestInstancePath, STR2 := '@');
AddTestNameToInstancePath := CONCAT(STR1 := CompleteTestInstancePath, STR2 := GVL_TcUnit.CurrentTestNameBeingCalled);
END_METHOD

METHOD PUBLIC AreAllTestsFinished : BOOL
VAR
    Counter : UINT;
    GetCurTaskIndex : GETCURTASKINDEX;
    NumberOfTestsToAnalyse : UINT(1..GVL_Param_TcUnit.MaxNumberOfTestsForEachTestSuite);
END_VAR
AreAllTestsFinished := FALSE;

IF NumberOfTests > 0 THEN
    AreAllTestsFinished := TRUE;
    // Limit the test analyse to the max array limit of 'Tests[]'
    NumberOfTestsToAnalyse := GetNumberOfTestsToAnalyse();
    // A test is considered finished if it is finished running (i.e. set by TEST_FINISHED) or if it is skipped/disabled
    FOR Counter := 1 TO NumberOfTestsToAnalyse BY 1 DO
        AreAllTestsFinished := AreAllTestsFinished AND (Tests[Counter].IsFinished() OR Tests[Counter].IsSkipped());
    END_FOR
END_IF

(* If we have been running at least one cycle and no tests are registered, it means that this testsuite is empty
   and doesn't contain any test cases. In that case, ignore this testsuite. *)
GetCurTaskIndex();
IF NumberOfTests = 0 AND NOT TwinCAT_SystemInfoVarList._TaskInfo[GetCurTaskIndex.index].FirstCycle AND StartedAt > 0 THEN
	AreAllTestsFinished := TRUE;
END_IF
END_METHOD

// Asserts that two LREAL 2D-arrays are equal to within a positive delta. If they are not, an assertion error is created.
METHOD PUBLIC AssertArray2dEquals_LREAL
VAR_IN_OUT
    Expecteds : ARRAY[*,*] OF LREAL; // LREAL 2d array with expected values
    Actuals : ARRAY[*,*] OF LREAL; // LREAL 2d array with actual values
END_VAR
VAR_INPUT
    Delta : LREAL; // The maximum delta between the value of expected and actual for which both numbers are still considered equal, proportional to the expected value in that array cell
    Message : T_MaxString; // The identifying message for the assertion error
END_VAR
VAR
    Equals : BOOL := TRUE;
    SizeEquals : BOOL := TRUE;
    ExpectedString : T_MaxString;
    ActualString : T_MaxString;
    AlreadyReported : BOOL;
    TestInstancePath : T_MaxString;
    DimensionIndex : USINT; // Index when looping through Dimensions
    LowerBoundExpecteds : ARRAY[1..2] OF DINT; // Lower bounds of Expecteds array in each dimension
    UpperBoundExpecteds : ARRAY[1..2] OF DINT; // Upper bounds of Expecteds array in each dimension
    LowerBoundActuals : ARRAY[1..2] OF DINT; // Lower bounds of Actuals array in each dimension
    UpperBoundActuals : ARRAY[1..2] OF DINT; // Upper bounds of Actuals array in each dimension
    SizeOfExpecteds : ARRAY[1..2] OF DINT; // Size of Expecteds array in each dimension
    SizeOfActuals : ARRAY[1..2] OF DINT; // Size of Actuals array in each dimension
    Offset : ARRAY[1..2] OF DINT; // Current Array index offsets from Lower Bound in each dimension
    ExpectedArrayIndex : ARRAY[1..2] OF DINT; // Array of current Expected array indexes when looping through arrays
    ActualArrayIndex : ARRAY[1..2] OF DINT; // Array of current Actual array indexes when looping through arrays
    Expected : LREAL; // Single expected value
    Actual : LREAL; // Single actual value
END_VAR
IF GVL_TcUnit.IgnoreCurrentTest OR GVL_TcUnit.CurrentTestIsFinished THEN
    RETURN;
END_IF

TestInstancePath := AddTestNameToInstancePath(FindTestSuiteInstancePath());

(* UPPER_BOUND and LOWER_BOUND require literals for their second parameter,
   so they can't be called in a dimension-based loop.
   Thus we copy the array dimensions into arrays which accept variable indexes *)
LowerBoundExpecteds[1] := LOWER_BOUND(Expecteds, 1);
UpperBoundExpecteds[1] := UPPER_BOUND(Expecteds, 1);
LowerBoundExpecteds[2] := LOWER_BOUND(Expecteds, 2);
UpperBoundExpecteds[2] := UPPER_BOUND(Expecteds, 2);
LowerBoundActuals[1] := LOWER_BOUND(Actuals, 1);
UpperBoundActuals[1] := UPPER_BOUND(Actuals, 1);
LowerBoundActuals[2] := LOWER_BOUND(Actuals, 2);
UpperBoundActuals[2] := UPPER_BOUND(Actuals, 2);

FOR DimensionIndex := 1 TO 2 DO
    SizeOfExpecteds[DimensionIndex] := ABS(UpperBoundExpecteds[DimensionIndex] - LowerBoundExpecteds[DimensionIndex]) + 1;
    SizeOfActuals[DimensionIndex] := ABS(UpperBoundActuals[DimensionIndex] - LowerBoundActuals[DimensionIndex]) + 1;

    IF SizeOfExpecteds[DimensionIndex] <> SizeOfActuals[DimensionIndex] THEN
        Equals := FALSE;
        SizeEquals := FALSE;
    END_IF
END_FOR

IF SizeEquals THEN
    (* Even though we know that both arrays are equal in size, the two arrays can start at two completely different
       indexes in each dimension, which needs to be taken into account. *)
    FOR Offset[1] := 0 TO SizeOfExpecteds[1] - 1 DO // Iterate Dimension 1
        FOR Offset[2] := 0 TO SizeOfExpecteds[2] - 1 DO // Iterate Dimension 2
            // Update index variables
            FOR DimensionIndex := 1 TO 2 DO
                ExpectedArrayIndex[DimensionIndex] := LowerBoundExpecteds[DimensionIndex] + Offset[DimensionIndex];
                ActualArrayIndex[DimensionIndex] := LowerBoundActuals[DimensionIndex] + Offset[DimensionIndex];
            END_FOR

            // Get array element values
            Expected := Expecteds[ExpectedArrayIndex[1], ExpectedArrayIndex[2]];
            Actual := Actuals[ActualArrayIndex[1], ActualArrayIndex[2]]; 

            IF ABS(Expected - Actual) > Delta THEN
                Equals := FALSE;
                EXIT;
            END_IF
        END_FOR

        // Check for loop bailout
        IF NOT Equals THEN
            EXIT;
        END_IF
    END_FOR
END_IF

AssertArrayResults.ReportResult(ExpectedsSize := DINT_TO_UDINT(SizeOfExpecteds[1] * SizeOfExpecteds[2]),
                                ExpectedsTypeClass := IBaseLibrary.TypeClass.TYPE_LREAL,
                                ActualsSize := DINT_TO_UDINT(SizeOfActuals[1] * SizeOfActuals[2]),
                                ActualsTypeClass := IBaseLibrary.TypeClass.TYPE_LREAL,
                                Message := Message,
                                TestInstancePath := TestInstancePath,
                                AlreadyReported => AlreadyReported);

IF NOT AlreadyReported AND NOT Equals THEN
    SetTestFailed(AssertionType := E_AssertionType.Type_Array2D_LREAL,
                  AssertionMessage := Message);

    IF NOT SizeEquals THEN
        Message := CONCAT(STR1 := Message, STR2 := ', size of arrays not matching.');
        ExpectedString := 'SIZE = [';
        ExpectedString := CONCAT(STR1 := ExpectedString,STR2 := DINT_TO_STRING(LowerBoundExpecteds[1]));
        ExpectedString := CONCAT(STR1 := ExpectedString, STR2 := '..');
        ExpectedString := CONCAT(STR1 := ExpectedString, STR2 := DINT_TO_STRING(UpperBoundExpecteds[1]));
        ExpectedString := CONCAT(STR1 := ExpectedString, STR2 := ',');
        ExpectedString := CONCAT(STR1 := ExpectedString, STR2 := DINT_TO_STRING(LowerBoundExpecteds[2]));
        ExpectedString := CONCAT(STR1 := ExpectedString, STR2 := '..');
        ExpectedString := CONCAT(STR1 := ExpectedString, STR2 := DINT_TO_STRING(UpperBoundExpecteds[2]));
        ExpectedString := CONCAT(STR1 := ExpectedString, STR2 := '] (');
        ExpectedString := CONCAT(STR1 := ExpectedString, STR2 := DINT_TO_STRING(SizeOfExpecteds[1]));
        ExpectedString := CONCAT(STR1 := ExpectedString, STR2 := 'x');
        ExpectedString := CONCAT(STR1 := ExpectedString, STR2 := DINT_TO_STRING(SizeOfExpecteds[2]));
        ExpectedString := CONCAT(STR1 := ExpectedString, STR2 := ')');

        ActualString := 'SIZE = [';
        ActualString := CONCAT(STR1 := ActualString, STR2 := DINT_TO_STRING(LowerBoundActuals[1]));
        ActualString := CONCAT(STR1 := ActualString, STR2 := '..');
        ActualString := CONCAT(STR1 := ActualString, STR2 := DINT_TO_STRING(UpperBoundActuals[1]));
        ActualString := CONCAT(STR1 := ActualString, STR2 := ',');
        ActualString := CONCAT(STR1 := ActualString, STR2 := DINT_TO_STRING(LowerBoundActuals[2]));
        ActualString := CONCAT(STR1 := ActualString, STR2 := '..');
        ActualString := CONCAT(STR1 := ActualString, STR2 := DINT_TO_STRING(UpperBoundActuals[2]));
        ActualString := CONCAT(STR1 := ActualString, STR2 := '] (');
        ActualString := CONCAT(STR1 := ActualString, STR2 := DINT_TO_STRING(SizeOfActuals[1]));
        ActualString := CONCAT(STR1 := ActualString, STR2 := 'x');
        ActualString := CONCAT(STR1 := ActualString, STR2 := DINT_TO_STRING(SizeOfActuals[2]));
        ActualString := CONCAT(STR1 := ActualString, STR2 := ')');
    ELSE
        ExpectedString := 'ARRAY[';
        ExpectedString := CONCAT(STR1 := ExpectedString, STR2 := DINT_TO_STRING(ExpectedArrayIndex[1]));
        ExpectedString := CONCAT(STR1 := ExpectedString, STR2 := ',');
        ExpectedString := CONCAT(STR1 := ExpectedString, STR2 := DINT_TO_STRING(ExpectedArrayIndex[2]));
        ExpectedString := CONCAT(STR1 := ExpectedString, STR2 := '] = ');
        ExpectedString := CONCAT(STR1 := ExpectedString, STR2 := LREAL_TO_STRING(Expected));

        ActualString := 'ARRAY[';
        ActualString := CONCAT(STR1 := ActualString, STR2 := DINT_TO_STRING(ActualArrayIndex[1]));
        ActualString := CONCAT(STR1 := ActualString, STR2 := ',');
        ActualString := CONCAT(STR1 := ActualString, STR2 := DINT_TO_STRING(ActualArrayIndex[2]));
        ActualString := CONCAT(STR1 := ActualString, STR2 := '] = ');
        ActualString := CONCAT(STR1 := ActualString, STR2 := LREAL_TO_STRING(Actual));
    END_IF

    AssertMessageFormatter.LogAssertFailure(Expected := ExpectedString,
                                            Actual := ActualString,
                                            Message := Message,
                                            TestInstancePath := TestInstancePath);
END_IF
END_METHOD

// Asserts that two REAL 2D-arrays are equal to within a positive delta. If they are not, an assertion error is created.
METHOD PUBLIC AssertArray2dEquals_REAL
VAR_IN_OUT
    Expecteds : ARRAY[*,*] OF REAL; // REAL 2d array with expected values
    Actuals : ARRAY[*,*] OF REAL; // REAL 2d array with actual values
END_VAR
VAR_INPUT
    Delta : REAL; // The maximum delta between the value of expected and actual for which both numbers are still considered equal, proportional to the expected value in that array cell
    Message : T_MaxString; // The identifying message for the assertion error
END_VAR
VAR
    Equals : BOOL := TRUE;
    SizeEquals : BOOL := TRUE;
    ExpectedString : T_MaxString;
    ActualString : T_MaxString;
    AlreadyReported : BOOL;
    TestInstancePath : T_MaxString;
    DimensionIndex : USINT; // Index when looping through Dimensions
    LowerBoundExpecteds : ARRAY[1..2] OF DINT; // Lower bounds of Expecteds array in each dimension
    UpperBoundExpecteds : ARRAY[1..2] OF DINT; // Upper bounds of Expecteds array in each dimension
    LowerBoundActuals : ARRAY[1..2] OF DINT; // Lower bounds of Actuals array in each dimension
    UpperBoundActuals : ARRAY[1..2] OF DINT; // Upper bounds of Actuals array in each dimension
    SizeOfExpecteds : ARRAY[1..2] OF DINT; // Size of Expecteds array in each dimension
    SizeOfActuals : ARRAY[1..2] OF DINT; // Size of Actuals array in each dimension
    Offset : ARRAY[1..2] OF DINT; // Current Array index offsets from Lower Bound in each dimension
    ExpectedArrayIndex : ARRAY[1..2] OF DINT; // Array of current Expected array indexes when looping through arrays
    ActualArrayIndex : ARRAY[1..2] OF DINT; // Array of current Actual array indexes when looping through arrays
    Expected : REAL; // Single expected value
    Actual : REAL; // Single actual value
END_VAR
IF GVL_TcUnit.IgnoreCurrentTest OR GVL_TcUnit.CurrentTestIsFinished THEN
    RETURN;
END_IF

TestInstancePath := AddTestNameToInstancePath(FindTestSuiteInstancePath());

(* UPPER_BOUND and LOWER_BOUND require literals for their second parameter, 
   so they can't be called in a dimension-based loop.
   Thus we copy the ARRAY dimensions into arrays which accept variable indexes *)
LowerBoundExpecteds[1] := LOWER_BOUND(Expecteds, 1);
UpperBoundExpecteds[1] := UPPER_BOUND(Expecteds, 1);
LowerBoundExpecteds[2] := LOWER_BOUND(Expecteds, 2);
UpperBoundExpecteds[2] := UPPER_BOUND(Expecteds, 2);
LowerBoundActuals[1] := LOWER_BOUND(Actuals, 1);
UpperBoundActuals[1] := UPPER_BOUND(Actuals, 1);
LowerBoundActuals[2] := LOWER_BOUND(Actuals, 2);
UpperBoundActuals[2] := UPPER_BOUND(Actuals, 2);

FOR DimensionIndex := 1 TO 2 DO
    SizeOfExpecteds[DimensionIndex] := ABS(UpperBoundExpecteds[DimensionIndex] - LowerBoundExpecteds[DimensionIndex]) + 1;
    SizeOfActuals[DimensionIndex] := ABS(UpperBoundActuals[DimensionIndex] - LowerBoundActuals[DimensionIndex]) + 1;

    IF SizeOfExpecteds[DimensionIndex] <> SizeOfActuals[DimensionIndex] THEN
        Equals := FALSE;
        SizeEquals := FALSE;
    END_IF
END_FOR

IF SizeEquals THEN
    (* Even though we know that both arrays are equal in size, the two arrays can start at two completely different
       indexes in each dimension, which needs to be taken into account. *)
    FOR Offset[1] := 0 TO SizeOfExpecteds[1] - 1 DO // Iterate Dimension 1
        FOR Offset[2] := 0 TO SizeOfExpecteds[2] - 1 DO // Iterate Dimension 2
            // Update index variables
            FOR DimensionIndex := 1 TO 2 DO
                ExpectedArrayIndex[DimensionIndex] := LowerBoundExpecteds[DimensionIndex] + Offset[DimensionIndex];
                ActualArrayIndex[DimensionIndex] := LowerBoundActuals[DimensionIndex] + Offset[DimensionIndex];
            END_FOR

            // Get array element values
            Expected := Expecteds[ExpectedArrayIndex[1], ExpectedArrayIndex[2]];
            Actual := Actuals[ActualArrayIndex[1], ActualArrayIndex[2]]; 

            IF ABS(Expected - Actual) > Delta THEN
                Equals := FALSE;
                EXIT;
            END_IF
        END_FOR

        // Check for loop bailout
        IF NOT Equals THEN
            EXIT;
        END_IF
    END_FOR
END_IF

AssertArrayResults.ReportResult(ExpectedsSize := DINT_TO_UDINT(SizeOfExpecteds[1] * SizeOfExpecteds[2]),
                                ExpectedsTypeClass := IBaseLibrary.TypeClass.TYPE_REAL,
                                ActualsSize := DINT_TO_UDINT(SizeOfActuals[1] * SizeOfActuals[2]),
                                ActualsTypeClass := IBaseLibrary.TypeClass.TYPE_REAL,
                                Message := Message,
                                TestInstancePath := TestInstancePath,
                                AlreadyReported => AlreadyReported);

IF NOT AlreadyReported AND NOT Equals THEN
    SetTestFailed(AssertionType := E_AssertionType.Type_Array2D_REAL,
                  AssertionMessage := Message);

    IF NOT SizeEquals THEN
        Message := CONCAT(STR1 := Message, STR2 := ', size of arrays not matching.');
        ExpectedString := 'SIZE = [';
        ExpectedString := CONCAT(STR1 := ExpectedString, STR2 := DINT_TO_STRING(LowerBoundExpecteds[1]));
        ExpectedString := CONCAT(STR1 := ExpectedString, STR2 := '..');
        ExpectedString := CONCAT(STR1 := ExpectedString, STR2 := DINT_TO_STRING(UpperBoundExpecteds[1]));
        ExpectedString := CONCAT(STR1 := ExpectedString, STR2 := ',');
        ExpectedString := CONCAT(STR1 := ExpectedString, STR2 := DINT_TO_STRING(LowerBoundExpecteds[2]));
        ExpectedString := CONCAT(STR1 := ExpectedString, STR2 := '..');
        ExpectedString := CONCAT(STR1 := ExpectedString, STR2 := DINT_TO_STRING(UpperBoundExpecteds[2]));
        ExpectedString := CONCAT(STR1 := ExpectedString, STR2 := '] (');
        ExpectedString := CONCAT(STR1 := ExpectedString, STR2 := DINT_TO_STRING(SizeOfExpecteds[1]));
        ExpectedString := CONCAT(STR1 := ExpectedString, STR2 := 'x');
        ExpectedString := CONCAT(STR1 := ExpectedString, STR2 := DINT_TO_STRING(SizeOfExpecteds[2]));
        ExpectedString := CONCAT(STR1 := ExpectedString, STR2 := ')');

        ActualString := 'SIZE = [';
        ActualString := CONCAT(STR1 := ActualString, STR2 := DINT_TO_STRING(LowerBoundActuals[1]));
        ActualString := CONCAT(STR1 := ActualString, STR2 := '..');
        ActualString := CONCAT(STR1 := ActualString, STR2 := DINT_TO_STRING(UpperBoundActuals[1]));
        ActualString := CONCAT(STR1 := ActualString, STR2 := ',');
        ActualString := CONCAT(STR1 := ActualString, STR2 := DINT_TO_STRING(LowerBoundActuals[2]));
        ActualString := CONCAT(STR1 := ActualString, STR2 := '..');
        ActualString := CONCAT(STR1 := ActualString, STR2 := DINT_TO_STRING(UpperBoundActuals[2]));
        ActualString := CONCAT(STR1 := ActualString, STR2 := '] (');
        ActualString := CONCAT(STR1 := ActualString, STR2 := DINT_TO_STRING(SizeOfActuals[1]));
        ActualString := CONCAT(STR1 := ActualString, STR2 := 'x');
        ActualString := CONCAT(STR1 := ActualString, STR2 := DINT_TO_STRING(SizeOfActuals[2]));
        ActualString := CONCAT(STR1 := ActualString, STR2 := ')');
    ELSE
        ExpectedString := 'ARRAY[';
        ExpectedString := CONCAT(STR1 := ExpectedString, STR2 := DINT_TO_STRING(ExpectedArrayIndex[1]));
        ExpectedString := CONCAT(STR1 := ExpectedString, STR2 := ',');
        ExpectedString := CONCAT(STR1 := ExpectedString, STR2 := DINT_TO_STRING(ExpectedArrayIndex[2]));
        ExpectedString := CONCAT(STR1 := ExpectedString, STR2 := '] = ');
        ExpectedString := CONCAT(STR1 := ExpectedString, STR2 := REAL_TO_STRING(Expected));

        ActualString := 'ARRAY[';
        ActualString := CONCAT(STR1 := ActualString, STR2 := DINT_TO_STRING(ActualArrayIndex[1]));
        ActualString := CONCAT(STR1 := ActualString, STR2 := ',');
        ActualString := CONCAT(STR1 := ActualString, STR2 := DINT_TO_STRING(ActualArrayIndex[2]));
        ActualString := CONCAT(STR1 := ActualString, STR2 := '] = ');
        ActualString := CONCAT(STR1 := ActualString, STR2 := REAL_TO_STRING(Actual));
    END_IF

    AssertMessageFormatter.LogAssertFailure(Expected := ExpectedString,
                                            Actual := ActualString,
                                            Message := Message,
                                            TestInstancePath := TestInstancePath);
END_IF
END_METHOD

// Asserts that two LREAL 3D-arrays are equal to within a positive delta. If they are not, an assertion error is created.
METHOD PUBLIC AssertArray3dEquals_LREAL
VAR_IN_OUT
    Expecteds : ARRAY[*,*,*] OF LREAL; // LREAL 3d array with expected values
    Actuals : ARRAY[*,*,*] OF LREAL; // LREAL 3d array with actual values
END_VAR
VAR_INPUT
    Delta : LREAL; // The maximum delta between the value of expected and actual for which both numbers are still considered equal, proportional to the expected value in that array cell
    Message : T_MaxString; // The identifying message for the assertion error
END_VAR
VAR
    Equals : BOOL := TRUE;
    SizeEquals : BOOL := TRUE;
    ExpectedString : T_MaxString;
    ActualString : T_MaxString;
    AlreadyReported : BOOL;
    TestInstancePath : T_MaxString;
    DimensionIndex : USINT;  // Index when looping through Dimensions
    LowerBoundExpecteds : ARRAY[1..3] OF DINT; // Lower bounds of Expecteds array in each dimension
    UpperBoundExpecteds : ARRAY[1..3] OF DINT; // Upper bounds of Expecteds array in each dimension
    LowerBoundActuals : ARRAY[1..3] OF DINT; // Lower bounds of Actuals array in each dimension
    UpperBoundActuals : ARRAY[1..3] OF DINT; // Upper bounds of Actuals array in each dimension
    SizeOfExpecteds : ARRAY[1..3] OF DINT; // Size of Expecteds array in each dimension
    SizeOfActuals : ARRAY[1..3] OF DINT; // Size of Actuals array in each dimension
    Offset : ARRAY[1..3] OF DINT; // Current Array index offsets from Lower Bound in each dimension
    ExpectedArrayIndex : ARRAY[1..3] OF DINT; // Array of current Expected array indexes when looping through arrays
    ActualArrayIndex : ARRAY[1..3] OF DINT; // Array of current Actual array indexes when looping through arrays
    Expected : LREAL; // Single expected value
    Actual : LREAL; // Single actual value
END_VAR
IF GVL_TcUnit.IgnoreCurrentTest OR GVL_TcUnit.CurrentTestIsFinished THEN
    RETURN;
END_IF

TestInstancePath := AddTestNameToInstancePath(FindTestSuiteInstancePath());

(* UPPER_BOUND and LOWER_BOUND require literals for their second parameter,
   so they can't be called in a dimension-based loop.
   Thus we copy the array dimensions into arrays which accept variable indexes *)
LowerBoundExpecteds[1] := LOWER_BOUND(Expecteds, 1);
UpperBoundExpecteds[1] := UPPER_BOUND(Expecteds, 1);
LowerBoundExpecteds[2] := LOWER_BOUND(Expecteds, 2);
UpperBoundExpecteds[2] := UPPER_BOUND(Expecteds, 2);
LowerBoundExpecteds[3] := LOWER_BOUND(Expecteds, 3);
UpperBoundExpecteds[3] := UPPER_BOUND(Expecteds, 3);
LowerBoundActuals[1] := LOWER_BOUND(Actuals, 1);
UpperBoundActuals[1] := UPPER_BOUND(Actuals, 1);
LowerBoundActuals[2] := LOWER_BOUND(Actuals, 2);
UpperBoundActuals[2] := UPPER_BOUND(Actuals, 2);
LowerBoundActuals[3] := LOWER_BOUND(Actuals, 3);
UpperBoundActuals[3] := UPPER_BOUND(Actuals, 3);

FOR DimensionIndex := 1 TO 3 DO
    SizeOfExpecteds[DimensionIndex] := ABS(UpperBoundExpecteds[DimensionIndex] - LowerBoundExpecteds[DimensionIndex]) + 1;
    SizeOfActuals[DimensionIndex] := ABS(UpperBoundActuals[DimensionIndex] - LowerBoundActuals[DimensionIndex]) + 1;

    IF SizeOfExpecteds[DimensionIndex] <> SizeOfActuals[DimensionIndex] THEN
        Equals := FALSE;
        SizeEquals := FALSE;
    END_IF
END_FOR

IF SizeEquals THEN
    (* Even though we know that both arrays are equal in size, the three arrays can start at three completely different
       indexes in each dimension, which needs to be taken into account. *)
    FOR Offset[1] := 0 TO SizeOfExpecteds[1] - 1 DO // Iterate Dimension 1
        FOR Offset[2] := 0 TO SizeOfExpecteds[2] - 1 DO // Iterate Dimension 2
            FOR Offset[3] := 0 TO SizeOfExpecteds[3] - 1 DO // Iterate Dimension 3
                // Update index variables
                FOR DimensionIndex := 1 TO 3 DO
                    ExpectedArrayIndex[DimensionIndex] := LowerBoundExpecteds[DimensionIndex] + Offset[DimensionIndex];
                    ActualArrayIndex[DimensionIndex] := LowerBoundActuals[DimensionIndex] + Offset[DimensionIndex];
                END_FOR

                // Get array element values
                Expected := Expecteds[ExpectedArrayIndex[1], ExpectedArrayIndex[2], ExpectedArrayIndex[3]];
                Actual := Actuals[ActualArrayIndex[1], ActualArrayIndex[2], ActualArrayIndex[3]]; 

                IF ABS(Expected - Actual) > Delta THEN
                    Equals := FALSE;
                    EXIT;
                END_IF
            END_FOR

            // Check for loop bailout
            IF NOT Equals THEN
                EXIT;
            END_IF
        END_FOR

        // Check for loop bailout
        IF NOT Equals THEN
            EXIT;
        END_IF
    END_FOR
END_IF

AssertArrayResults.ReportResult(ExpectedsSize := DINT_TO_UDINT(SizeOfExpecteds[1] * SizeOfExpecteds[2] * SizeOfExpecteds[3]),
                                ExpectedsTypeClass := IBaseLibrary.TypeClass.TYPE_LREAL,
                                ActualsSize := DINT_TO_UDINT(SizeOfActuals[1] * SizeOfActuals[2] * SizeOfActuals[3]),
                                ActualsTypeClass := IBaseLibrary.TypeClass.TYPE_LREAL,
                                Message := Message,
                                TestInstancePath := TestInstancePath,
                                AlreadyReported => AlreadyReported);

IF NOT AlreadyReported AND NOT Equals THEN
    SetTestFailed(AssertionType := E_AssertionType.Type_Array3D_LREAL,
                  AssertionMessage := Message);

    IF NOT SizeEquals THEN
        Message := CONCAT(STR1 := Message, STR2 := ', size of arrays not matching.');
        ExpectedString := 'SIZE = [';
        ExpectedString := CONCAT(STR1 := ExpectedString, STR2 := DINT_TO_STRING(LowerBoundExpecteds[1]));
        ExpectedString := CONCAT(STR1 := ExpectedString, STR2 := '..');
        ExpectedString := CONCAT(STR1 := ExpectedString, STR2 := DINT_TO_STRING(UpperBoundExpecteds[1]));
        ExpectedString := CONCAT(STR1 := ExpectedString, STR2 := ',');
        ExpectedString := CONCAT(STR1 := ExpectedString, STR2 := DINT_TO_STRING(LowerBoundExpecteds[2]));
        ExpectedString := CONCAT(STR1 := ExpectedString, STR2 := '..');
        ExpectedString := CONCAT(STR1 := ExpectedString, STR2 := DINT_TO_STRING(UpperBoundExpecteds[2]));
        ExpectedString := CONCAT(STR1 := ExpectedString, STR2 := ',');
        ExpectedString := CONCAT(STR1 := ExpectedString, STR2 := DINT_TO_STRING(LowerBoundExpecteds[3]));
        ExpectedString := CONCAT(STR1 := ExpectedString, STR2 := '..');
        ExpectedString := CONCAT(STR1 := ExpectedString, STR2 := DINT_TO_STRING(UpperBoundExpecteds[3]));
        ExpectedString := CONCAT(STR1 := ExpectedString, STR2 := '] (');
        ExpectedString := CONCAT(STR1 := ExpectedString, STR2 := DINT_TO_STRING(SizeOfExpecteds[1]));
        ExpectedString := CONCAT(STR1 := ExpectedString, STR2 := 'x');
        ExpectedString := CONCAT(STR1 := ExpectedString, STR2 := DINT_TO_STRING(SizeOfExpecteds[2]));
        ExpectedString := CONCAT(STR1 := ExpectedString, STR2 := 'x');
        ExpectedString := CONCAT(STR1 := ExpectedString, STR2 := DINT_TO_STRING(SizeOfExpecteds[3]));
        ExpectedString := CONCAT(STR1 := ExpectedString, STR2 := ')');

        ActualString := 'SIZE = [';
        ActualString := CONCAT(STR1 := ActualString, STR2 := DINT_TO_STRING(LowerBoundActuals[1]));
        ActualString := CONCAT(STR1 := ActualString, STR2 := '..');
        ActualString := CONCAT(STR1 := ActualString, STR2 := DINT_TO_STRING(UpperBoundActuals[1]));
        ActualString := CONCAT(STR1 := ActualString, STR2 := ',');
        ActualString := CONCAT(STR1 := ActualString, STR2 := DINT_TO_STRING(LowerBoundActuals[2]));
        ActualString := CONCAT(STR1 := ActualString, STR2 := '..');
        ActualString := CONCAT(STR1 := ActualString, STR2 := DINT_TO_STRING(UpperBoundActuals[2]));
        ActualString := CONCAT(STR1 := ActualString, STR2 := ',');
        ActualString := CONCAT(STR1 := ActualString, STR2 := DINT_TO_STRING(LowerBoundActuals[3]));
        ActualString := CONCAT(STR1 := ActualString, STR2 := '..');
        ActualString := CONCAT(STR1 := ActualString, STR2 := DINT_TO_STRING(UpperBoundActuals[3]));
        ActualString := CONCAT(STR1 := ActualString, STR2 := '] (');
        ActualString := CONCAT(STR1 := ActualString, STR2 := DINT_TO_STRING(SizeOfActuals[1]));
        ActualString := CONCAT(STR1 := ActualString, STR2 := 'x');
        ActualString := CONCAT(STR1 := ActualString, STR2 := DINT_TO_STRING(SizeOfActuals[2]));
        ActualString := CONCAT(STR1 := ActualString, STR2 := 'x');
        ActualString := CONCAT(STR1 := ActualString, STR2 := DINT_TO_STRING(SizeOfActuals[3]));
        ActualString := CONCAT(STR1 := ActualString, STR2 := ')');
    ELSE
        ExpectedString := 'ARRAY[';
        ExpectedString := CONCAT(STR1 := ExpectedString, STR2 := DINT_TO_STRING(ExpectedArrayIndex[1]));
        ExpectedString := CONCAT(STR1 := ExpectedString, STR2 := ',');
        ExpectedString := CONCAT(STR1 := ExpectedString, STR2 := DINT_TO_STRING(ExpectedArrayIndex[2]));
        ExpectedString := CONCAT(STR1 := ExpectedString, STR2 := ',');
        ExpectedString := CONCAT(STR1 := ExpectedString, STR2 := DINT_TO_STRING(ExpectedArrayIndex[3]));
        ExpectedString := CONCAT(STR1 := ExpectedString, STR2 := '] = ');
        ExpectedString := CONCAT(STR1 := ExpectedString, STR2 := LREAL_TO_STRING(Expected) );

        ActualString := 'ARRAY[';
        ActualString := CONCAT(STR1 := ActualString, STR2 := DINT_TO_STRING(ActualArrayIndex[1]));
        ActualString := CONCAT(STR1 := ActualString, STR2 := ',');
        ActualString := CONCAT(STR1 := ActualString, STR2 := DINT_TO_STRING(ActualArrayIndex[2]));
        ActualString := CONCAT(STR1 := ActualString, STR2 := ',');
        ActualString := CONCAT(STR1 := ActualString, STR2 := DINT_TO_STRING(ActualArrayIndex[3]));
        ActualString := CONCAT(STR1 := ActualString, STR2 := '] = ');
        ActualString := CONCAT(STR1 := ActualString, STR2 := LREAL_TO_STRING(Actual));
    END_IF

    AssertMessageFormatter.LogAssertFailure(Expected := ExpectedString,
                                            Actual := ActualString,
                                            Message := Message,
                                            TestInstancePath := TestInstancePath);
END_IF
END_METHOD

// Asserts that two REAL 3D-arrays are equal to within a positive delta. If they are not, an assertion error is created.
METHOD PUBLIC AssertArray3dEquals_REAL
VAR_IN_OUT
    Expecteds : ARRAY[*,*,*] OF REAL; // REAL 3d array with expected values
    Actuals : ARRAY[*,*,*] OF REAL; // REAL 3d array with actual values
END_VAR
VAR_INPUT
    Delta : REAL; // The maximum delta between the value of expected and actual for which both numbers are still considered equal, proportional to the expected value in that array cell
    Message : T_MaxString; // The identifying message for the assertion error
END_VAR
VAR
    Equals : BOOL := TRUE;
    SizeEquals : BOOL := TRUE;
    ExpectedString : T_MaxString;
    ActualString : T_MaxString;
    AlreadyReported : BOOL;
    TestInstancePath : T_MaxString;
    DimensionIndex : USINT;  // Index when looping through Dimensions
    LowerBoundExpecteds : ARRAY[1..3] OF DINT; // Lower bounds of Expecteds array in each dimension
    UpperBoundExpecteds : ARRAY[1..3] OF DINT; // Upper bounds of Expecteds array in each dimension
    LowerBoundActuals : ARRAY[1..3] OF DINT; // Lower bounds of Actuals array in each dimension
    UpperBoundActuals : ARRAY[1..3] OF DINT; // Upper bounds of Actuals array in each dimension
    SizeOfExpecteds : ARRAY[1..3] OF DINT; // Size of Expecteds array in each dimension
    SizeOfActuals : ARRAY[1..3] OF DINT; // Size of Actuals array in each dimension
    Offset : ARRAY[1..3] OF DINT; // Current Array index offsets from Lower Bound in each dimension
    ExpectedArrayIndex : ARRAY[1..3] OF DINT; // Array of current Expected array indexes when looping through arrays
    ActualArrayIndex : ARRAY[1..3] OF DINT; // Array of current Actual array indexes when looping through arrays
    Expected : REAL; // Single expected value
    Actual : REAL; // Single actual value
    ExpectedValueString : T_MaxString;
    ActualValueString : T_MaxString;
    FormatString : FB_FormatString; // String formatter for output messages
END_VAR
IF GVL_TcUnit.IgnoreCurrentTest OR GVL_TcUnit.CurrentTestIsFinished THEN
    RETURN;
END_IF

TestInstancePath := AddTestNameToInstancePath(FindTestSuiteInstancePath());

(* UPPER_BOUND and LOWER_BOUND require literals for their second parameter,
   so they can't be called in a dimension-based loop.
   Thus we copy the array dimensions into arrays which accept variable indexes *)
LowerBoundExpecteds[1] := LOWER_BOUND(Expecteds, 1);
UpperBoundExpecteds[1] := UPPER_BOUND(Expecteds, 1);
LowerBoundExpecteds[2] := LOWER_BOUND(Expecteds, 2);
UpperBoundExpecteds[2] := UPPER_BOUND(Expecteds, 2);
LowerBoundExpecteds[3] := LOWER_BOUND(Expecteds, 3);
UpperBoundExpecteds[3] := UPPER_BOUND(Expecteds, 3);
LowerBoundActuals[1] := LOWER_BOUND(Actuals, 1);
UpperBoundActuals[1] := UPPER_BOUND(Actuals, 1);
LowerBoundActuals[2] := LOWER_BOUND(Actuals, 2);
UpperBoundActuals[2] := UPPER_BOUND(Actuals, 2);
LowerBoundActuals[3] := LOWER_BOUND(Actuals, 3);
UpperBoundActuals[3] := UPPER_BOUND(Actuals, 3);

FOR DimensionIndex := 1 TO 3 DO
    SizeOfExpecteds[DimensionIndex] := ABS(UpperBoundExpecteds[DimensionIndex] - LowerBoundExpecteds[DimensionIndex]) + 1;
    SizeOfActuals[DimensionIndex] := ABS(UpperBoundActuals[DimensionIndex] - LowerBoundActuals[DimensionIndex]) + 1;

    IF SizeOfExpecteds[DimensionIndex] <> SizeOfActuals[DimensionIndex] THEN
        Equals := FALSE;
        SizeEquals := FALSE;
    END_IF
END_FOR

IF SizeEquals THEN
    (* Even though we know that both arrays are equal in size, the two arrays can start at two completely different
       indexes in each dimension, which needs to be taken into account. *)
    FOR Offset[1] := 0 TO SizeOfExpecteds[1] - 1 DO // Iterate Dimension 1
        FOR Offset[2] := 0 TO SizeOfExpecteds[2] - 1 DO // Iterate Dimension 2
            FOR Offset[3] := 0 TO SizeOfExpecteds[3] - 1 DO // Iterate Dimension 3
                // Update index variables
                FOR DimensionIndex := 1 TO 3 DO
                    ExpectedArrayIndex[DimensionIndex] := LowerBoundExpecteds[DimensionIndex] + Offset[DimensionIndex];
                    ActualArrayIndex[DimensionIndex] := LowerBoundActuals[DimensionIndex] + Offset[DimensionIndex];
                END_FOR

                // Get array element values
                Expected := Expecteds[ExpectedArrayIndex[1], ExpectedArrayIndex[2], ExpectedArrayIndex[3]];
                Actual := Actuals[ActualArrayIndex[1], ActualArrayIndex[2], ActualArrayIndex[3]]; 

                IF ABS(Expected - Actual) > Delta THEN
                    Equals := FALSE;
                    EXIT;
                END_IF
            END_FOR

            // Check for loop bailout
            IF NOT Equals THEN
                EXIT;
            END_IF
        END_FOR

        // Check for loop bailout
        IF NOT Equals THEN
            EXIT;
        END_IF
    END_FOR
END_IF

AssertArrayResults.ReportResult(ExpectedsSize := DINT_TO_UDINT(SizeOfExpecteds[1] * SizeOfExpecteds[2] * SizeOfExpecteds[3]),
                                ExpectedsTypeClass := IBaseLibrary.TypeClass.TYPE_REAL,
                                ActualsSize := DINT_TO_UDINT(SizeOfActuals[1] * SizeOfActuals[2] * SizeOfActuals[3]),
                                ActualsTypeClass := IBaseLibrary.TypeClass.TYPE_REAL,
                                Message := Message,
                                TestInstancePath := TestInstancePath,
                                AlreadyReported => AlreadyReported);

IF NOT AlreadyReported AND NOT Equals THEN
    SetTestFailed(AssertionType := E_AssertionType.Type_Array3D_REAL,
                  AssertionMessage := Message);

    IF NOT SizeEquals THEN
        Message := CONCAT(STR1 := Message, STR2 := ', size of arrays not matching.');
        ExpectedString := 'SIZE = [';
        ExpectedString := CONCAT(STR1 := ExpectedString, STR2 := DINT_TO_STRING(LowerBoundExpecteds[1]));
        ExpectedString := CONCAT(STR1 := ExpectedString, STR2 := '..');
        ExpectedString := CONCAT(STR1 := ExpectedString, STR2 := DINT_TO_STRING(UpperBoundExpecteds[1]));
        ExpectedString := CONCAT(STR1 := ExpectedString, STR2 := ',');
        ExpectedString := CONCAT(STR1 := ExpectedString, STR2 := DINT_TO_STRING(LowerBoundExpecteds[2]));
        ExpectedString := CONCAT(STR1 := ExpectedString, STR2 := '..');
        ExpectedString := CONCAT(STR1 := ExpectedString, STR2 := DINT_TO_STRING(UpperBoundExpecteds[2]));
        ExpectedString := CONCAT(STR1 := ExpectedString, STR2 := ',');
        ExpectedString := CONCAT(STR1 := ExpectedString, STR2 := DINT_TO_STRING(LowerBoundExpecteds[3]));
        ExpectedString := CONCAT(STR1 := ExpectedString, STR2 := '..');
        ExpectedString := CONCAT(STR1 := ExpectedString, STR2 := DINT_TO_STRING(UpperBoundExpecteds[3]));
        ExpectedString := CONCAT(STR1 := ExpectedString, STR2 := '] (');
        ExpectedString := CONCAT(STR1 := ExpectedString, STR2 := DINT_TO_STRING(SizeOfExpecteds[1]));
        ExpectedString := CONCAT(STR1 := ExpectedString, STR2 := 'x');
        ExpectedString := CONCAT(STR1 := ExpectedString, STR2 := DINT_TO_STRING(SizeOfExpecteds[2]));
        ExpectedString := CONCAT(STR1 := ExpectedString, STR2 := 'x');
        ExpectedString := CONCAT(STR1 := ExpectedString, STR2 := DINT_TO_STRING(SizeOfExpecteds[3]));
        ExpectedString := CONCAT(STR1 := ExpectedString, STR2 := ')');

        ActualString := 'SIZE = [';
        ActualString := CONCAT(STR1 := ActualString, STR2 := DINT_TO_STRING(LowerBoundActuals[1]));
        ActualString := CONCAT(STR1 := ActualString, STR2 := '..');
        ActualString := CONCAT(STR1 := ActualString, STR2 := DINT_TO_STRING(UpperBoundActuals[1]));
        ActualString := CONCAT(STR1 := ActualString, STR2 := ',');
        ActualString := CONCAT(STR1 := ActualString, STR2 := DINT_TO_STRING(LowerBoundActuals[2]));
        ActualString := CONCAT(STR1 := ActualString, STR2 := '..');
        ActualString := CONCAT(STR1 := ActualString, STR2 := DINT_TO_STRING(UpperBoundActuals[2]));
        ActualString := CONCAT(STR1 := ActualString, STR2 := ',');
        ActualString := CONCAT(STR1 := ActualString, STR2 := DINT_TO_STRING(LowerBoundActuals[3]));
        ActualString := CONCAT(STR1 := ActualString, STR2 := '..');
        ActualString := CONCAT(STR1 := ActualString, STR2 := DINT_TO_STRING(UpperBoundActuals[3]));
        ActualString := CONCAT(STR1 := ActualString, STR2 := '] (');
        ActualString := CONCAT(STR1 := ActualString, STR2 := DINT_TO_STRING(SizeOfActuals[1]));
        ActualString := CONCAT(STR1 := ActualString, STR2 := 'x');
        ActualString := CONCAT(STR1 := ActualString, STR2 := DINT_TO_STRING(SizeOfActuals[2]));
        ActualString := CONCAT(STR1 := ActualString, STR2 := 'x');
        ActualString := CONCAT(STR1 := ActualString, STR2 := DINT_TO_STRING(SizeOfActuals[3]));
        ActualString := CONCAT(STR1 := ActualString, STR2 := ')');
    ELSE
        ExpectedString := 'ARRAY[';
        ExpectedString := CONCAT(STR1 := ExpectedString, STR2 := DINT_TO_STRING(ExpectedArrayIndex[1]));
        ExpectedString := CONCAT(STR1 := ExpectedString, STR2 := ',');
        ExpectedString := CONCAT(STR1 := ExpectedString, STR2 := DINT_TO_STRING(ExpectedArrayIndex[2]));
        ExpectedString := CONCAT(STR1 := ExpectedString, STR2 := ',');
        ExpectedString := CONCAT(STR1 := ExpectedString, STR2 := DINT_TO_STRING(ExpectedArrayIndex[3]));
        ExpectedString := CONCAT(STR1 := ExpectedString, STR2 := '] = ');
        ExpectedString := CONCAT(STR1 := ExpectedString, STR2 := REAL_TO_STRING(Expected) );

        ActualString := 'ARRAY[';
        ActualString := CONCAT(STR1 := ActualString, STR2 := DINT_TO_STRING(ActualArrayIndex[1]));
        ActualString := CONCAT(STR1 := ActualString, STR2 := ',');
        ActualString := CONCAT(STR1 := ActualString, STR2 := DINT_TO_STRING(ActualArrayIndex[2]));
        ActualString := CONCAT(STR1 := ActualString, STR2 := ',');
        ActualString := CONCAT(STR1 := ActualString, STR2 := DINT_TO_STRING(ActualArrayIndex[3]));
        ActualString := CONCAT(STR1 := ActualString, STR2 := '] = ');
        ActualString := CONCAT(STR1 := ActualString, STR2 := REAL_TO_STRING(Actual));
    END_IF

    AssertMessageFormatter.LogAssertFailure(Expected := ExpectedString,
                                            Actual := ActualString,
                                            Message := Message,
                                            TestInstancePath := TestInstancePath);
END_IF
END_METHOD

// Asserts that two BOOL arrays are equal. If they are not, an assertion error is created.
METHOD PUBLIC AssertArrayEquals_BOOL
VAR_IN_OUT
    Expecteds : ARRAY[*] OF BOOL; // BOOL array with expected values
    Actuals : ARRAY[*] OF BOOL; // BOOL array with actual values
END_VAR
VAR_INPUT
    Message : T_MaxString; // The identifying message for the assertion error
END_VAR
VAR
    Equals : BOOL := TRUE;
    SizeEquals : BOOL := TRUE;
    Index : DINT;
    ExpectedString : T_MaxString;
    ActualString : T_MaxString;
    AlreadyReported : BOOL;
    TestInstancePath : T_MaxString;
    SizeOfExpecteds : DINT;
    SizeOfActuals : DINT;
    ExpectedsIndex : DINT;
    ActualsIndex : DINT;
END_VAR
IF GVL_TcUnit.IgnoreCurrentTest OR GVL_TcUnit.CurrentTestIsFinished THEN
    RETURN;
END_IF

TestInstancePath := AddTestNameToInstancePath(FindTestSuiteInstancePath());

SizeOfExpecteds := ABS(UPPER_BOUND(Expecteds, 1) - LOWER_BOUND(Expecteds, 1)) + 1;
SizeOfActuals := ABS(UPPER_BOUND(Actuals, 1) - LOWER_BOUND(Actuals, 1)) + 1;

IF SizeOfExpecteds <> SizeOfActuals THEN
    Equals := FALSE;
    SizeEquals := FALSE;
ELSE
    (* Even though we know that both arrays are equal in size, the two arrays can start at two completely different
       indexes, which needs to be taken into account for. *)
    ExpectedsIndex := LOWER_BOUND(Expecteds, 1); // The start position for the expecteds
    ActualsIndex := LOWER_BOUND(Actuals, 1); // The start position for the actuals
    FOR Index := 1 TO SizeOfExpecteds BY 1 DO
        IF Expecteds[ExpectedsIndex] <> Actuals[ActualsIndex] THEN
            Equals := FALSE;
            EXIT;
        END_IF
        ExpectedsIndex := ExpectedsIndex + 1;
        ActualsIndex := ActualsIndex + 1;
    END_FOR
END_IF

AssertArrayResults.ReportResult(ExpectedsSize := DINT_TO_UDINT(SizeOfExpecteds),
                                ExpectedsTypeClass := IBaseLibrary.TypeClass.TYPE_BOOL,
                                ActualsSize := DINT_TO_UDINT(SizeOfActuals),
                                ActualsTypeClass := IBaseLibrary.TypeClass.TYPE_BOOL,
                                Message := Message,
                                TestInstancePath := TestInstancePath,
                                AlreadyReported => AlreadyReported);

IF NOT AlreadyReported AND NOT Equals THEN
    SetTestFailed(AssertionType := E_AssertionType.Type_Array_BOOL,
                  AssertionMessage := Message);

    IF NOT SizeEquals THEN
        Message := CONCAT(STR1 := Message, STR2 := ', size of arrays not matching.');
        ExpectedString := 'SIZE = ';
        ExpectedString := CONCAT(STR1 := ExpectedString, STR2 := DINT_TO_STRING(SizeOfExpecteds));
        ActualString := 'SIZE = ';
        ActualString := CONCAT(STR1 := ActualString, STR2 := DINT_TO_STRING(SizeOfActuals));
    ELSE
        ExpectedString := 'ARRAY[';
        ExpectedString := CONCAT(STR1 := ExpectedString, STR2 := DINT_TO_STRING(ExpectedsIndex));
        ExpectedString := CONCAT(STR1 := ExpectedString, STR2 := '] = ');
        ExpectedString := CONCAT(STR1 := ExpectedString, STR2 := BOOL_TO_STRING(Expecteds[ExpectedsIndex]));

        ActualString := 'ARRAY[';
        ActualString := CONCAT(STR1 := ActualString, STR2 := DINT_TO_STRING(ActualsIndex));
        ActualString := CONCAT(STR1 := ActualString, STR2 := '] = ');
        ActualString := CONCAT(STR1 := ActualString, STR2 := BOOL_TO_STRING(Actuals[ActualsIndex]));
    END_IF

    AssertMessageFormatter.LogAssertFailure(Expected := ExpectedString,
                                            Actual := ActualString,
                                            Message := Message,
                                            TestInstancePath := TestInstancePath);
END_IF
END_METHOD

// Asserts that two BYTE arrays are equal. If they are not, an assertion error is created.
METHOD PUBLIC AssertArrayEquals_BYTE
VAR_IN_OUT
    Expecteds : ARRAY[*] OF BYTE; // BYTE array with expected values
    Actuals : ARRAY[*] OF BYTE; // BYTE array with actual values
END_VAR
VAR_INPUT
    Message : T_MaxString; // The identifying message for the assertion error
END_VAR
VAR
    Equals : BOOL := TRUE;
    SizeEquals : BOOL := TRUE;
    Index : DINT;
    ExpectedString : T_MaxString;
    ActualString : T_MaxString;
    AlreadyReported : BOOL;
    TestInstancePath : T_MaxString;
    SizeOfExpecteds : DINT;
    SizeOfActuals : DINT;
    ExpectedByteString : STRING;
    ActualByteString : STRING;
    ExpectedsIndex : DINT;
    ActualsIndex : DINT;
END_VAR
IF GVL_TcUnit.IgnoreCurrentTest OR GVL_TcUnit.CurrentTestIsFinished THEN
    RETURN;
END_IF

TestInstancePath := AddTestNameToInstancePath(FindTestSuiteInstancePath());

SizeOfExpecteds := ABS(UPPER_BOUND(Expecteds, 1) - LOWER_BOUND(Expecteds, 1)) + 1;
SizeOfActuals := ABS(UPPER_BOUND(Actuals, 1) - LOWER_BOUND(Actuals, 1)) + 1;

IF SizeOfExpecteds <> SizeOfActuals THEN
    Equals := FALSE;
    SizeEquals := FALSE;
ELSE
    (* Even though we know that both arrays are equal in size, the two arrays can start at two completely different
       indexes, which needs to be taken into account for. *)
    ExpectedsIndex := LOWER_BOUND(Expecteds, 1); // The start position for the expecteds
    ActualsIndex := LOWER_BOUND(Actuals, 1); // The start position for the actuals
    FOR Index := 1 TO SizeOfExpecteds BY 1 DO
        IF Expecteds[ExpectedsIndex] <> Actuals[ActualsIndex] THEN
            Equals := FALSE;
            EXIT;
        END_IF
        ExpectedsIndex := ExpectedsIndex + 1;
        ActualsIndex := ActualsIndex + 1;
    END_FOR
END_IF


AssertArrayResults.ReportResult(ExpectedsSize := DINT_TO_UDINT(SizeOfExpecteds),
                                ExpectedsTypeClass := IBaseLibrary.TypeClass.TYPE_BYTE,
                                ActualsSize := DINT_TO_UDINT(SizeOfActuals),
                                ActualsTypeClass := IBaseLibrary.TypeClass.TYPE_BYTE,
                                Message := Message,
                                TestInstancePath := TestInstancePath,
                                AlreadyReported => AlreadyReported);

IF NOT AlreadyReported AND NOT Equals THEN
    SetTestFailed(AssertionType := E_AssertionType.Type_Array_BYTE,
                  AssertionMessage := Message);
    
    IF NOT SizeEquals THEN
        Message := CONCAT(STR1 := Message, STR2 := ', size of arrays not matching.');
        ExpectedString := 'SIZE = ';
        ExpectedString := CONCAT(STR1 := ExpectedString, STR2 := DINT_TO_STRING(SizeOfExpecteds));
        ActualString := 'SIZE = ';
        ActualString := CONCAT(STR1 := ActualString, STR2 := DINT_TO_STRING(SizeOfActuals));
    ELSE
        ExpectedByteString := CONCAT(STR1 := '0x',
                                                  STR2 := BYTE_TO_HEXSTR(in := Expecteds[ExpectedsIndex],
                                                                                       iPrecision := 2,
                                                                                       bLoCase := FALSE));
        ExpectedString := 'ARRAY[';
        ExpectedString := CONCAT(STR1 := ExpectedString, STR2 := DINT_TO_STRING(ExpectedsIndex));
        ExpectedString := CONCAT(STR1 := ExpectedString, STR2 := '] = ');
        ExpectedString := CONCAT(STR1 := ExpectedString, STR2 := ExpectedByteString);

        ActualByteString := CONCAT(STR1 := '0x',
                                                STR2 := BYTE_TO_HEXSTR(in := Actuals[ActualsIndex],
                                                                                     iPrecision := 2,
                                                                                     bLoCase := FALSE));
        ActualString := 'ARRAY[';
        ActualString := CONCAT(STR1 := ActualString, STR2 := DINT_TO_STRING(ActualsIndex));
        ActualString := CONCAT(STR1 := ActualString, STR2 := '] = ');
        ActualString := CONCAT(STR1 := ActualString, STR2 := ActualByteString);
    END_IF

    AssertMessageFormatter.LogAssertFailure(Expected := ExpectedString,
                                            Actual := ActualString,
                                            Message := Message,
                                            TestInstancePath := TestInstancePath);
END_IF
END_METHOD

// Asserts that two DINT arrays are equal. If they are not, an assertion error is created.
METHOD PUBLIC AssertArrayEquals_DINT
VAR_IN_OUT
    Expecteds : ARRAY[*] OF DINT; // DINT array with expected values
    Actuals : ARRAY[*] OF DINT; // DINT array with actual values
END_VAR
VAR_INPUT
    Message : T_MaxString; // The identifying message for the assertion error
END_VAR
VAR
    Equals : BOOL := TRUE;
    SizeEquals : BOOL := TRUE;
    Index : DINT;
    ExpectedString : T_MaxString;
    ActualString : T_MaxString;
    AlreadyReported : BOOL;
    TestInstancePath : T_MaxString;
    SizeOfExpecteds : DINT;
    SizeOfActuals : DINT;
    ExpectedsIndex : DINT;
    ActualsIndex : DINT;
END_VAR
IF GVL_TcUnit.IgnoreCurrentTest OR GVL_TcUnit.CurrentTestIsFinished THEN
    RETURN;
END_IF

TestInstancePath := AddTestNameToInstancePath(FindTestSuiteInstancePath());

SizeOfExpecteds := ABS(UPPER_BOUND(Expecteds, 1) - LOWER_BOUND(Expecteds, 1)) + 1;
SizeOfActuals := ABS(UPPER_BOUND(Actuals, 1) - LOWER_BOUND(Actuals, 1)) + 1;

IF SizeOfExpecteds <> SizeOfActuals THEN
    Equals := FALSE;
    SizeEquals := FALSE;
ELSE
    (* Even though we know that both arrays are equal in size, the two arrays can start at two completely different
       indexes, which needs to be taken into account for. *)
    ExpectedsIndex := LOWER_BOUND(Expecteds, 1); // The start position for the expecteds
    ActualsIndex := LOWER_BOUND(Actuals, 1); // The start position for the actuals
    FOR Index := 1 TO SizeOfExpecteds BY 1 DO
        IF Expecteds[ExpectedsIndex] <> Actuals[ActualsIndex] THEN
            Equals := FALSE;
            EXIT;
        END_IF
        ExpectedsIndex := ExpectedsIndex + 1;
        ActualsIndex := ActualsIndex + 1;
    END_FOR
END_IF

AssertArrayResults.ReportResult(ExpectedsSize := DINT_TO_UDINT(SizeOfExpecteds),
                                ExpectedsTypeClass := IBaseLibrary.TypeClass.TYPE_DINT,
                                ActualsSize := DINT_TO_UDINT(SizeOfActuals),
                                ActualsTypeClass := IBaseLibrary.TypeClass.TYPE_DINT,
                                Message := Message,
                                TestInstancePath := TestInstancePath,
                                AlreadyReported => AlreadyReported);

IF NOT AlreadyReported AND NOT Equals THEN
    SetTestFailed(AssertionType := E_AssertionType.Type_Array_DINT,
                  AssertionMessage := Message);

    IF NOT SizeEquals THEN
        Message := CONCAT(STR1 := Message, STR2 := ', size of arrays not matching.');
        ExpectedString := 'SIZE = ';
        ExpectedString := CONCAT(STR1 := ExpectedString, STR2 := DINT_TO_STRING(SizeOfExpecteds));
        ActualString := 'SIZE = ';
        ActualString := CONCAT(STR1 := ActualString, STR2 := DINT_TO_STRING(SizeOfActuals));
    ELSE
        ExpectedString := 'ARRAY[';
        ExpectedString := CONCAT(STR1 := ExpectedString, STR2 := DINT_TO_STRING(ExpectedsIndex));
        ExpectedString := CONCAT(STR1 := ExpectedString, STR2 := '] = ');
        ExpectedString := CONCAT(STR1 := ExpectedString, STR2 := DINT_TO_STRING(Expecteds[ExpectedsIndex]));

        ActualString := 'ARRAY[';
        ActualString := CONCAT(STR1 := ActualString, STR2 := DINT_TO_STRING(ActualsIndex));
        ActualString := CONCAT(STR1 := ActualString, STR2 := '] = ');
        ActualString := CONCAT(STR1 := ActualString, STR2 := DINT_TO_STRING(Actuals[ActualsIndex]));
    END_IF

    AssertMessageFormatter.LogAssertFailure(Expected := ExpectedString,
                                            Actual := ActualString,
                                            Message := Message,
                                            TestInstancePath := TestInstancePath);
END_IF
END_METHOD

// Asserts that two DWORD arrays are equal. If they are not, an assertion error is created.
METHOD PUBLIC AssertArrayEquals_DWORD
VAR_IN_OUT
    Expecteds : ARRAY[*] OF DWORD; // DWORD array with expected values
    Actuals : ARRAY[*] OF DWORD; // DWORD array with actual values
END_VAR
VAR_INPUT
    Message : T_MaxString; // The identifying message for the assertion error
END_VAR
VAR
    Equals : BOOL := TRUE;
    SizeEquals : BOOL := TRUE;
    Index : DINT;
    ExpectedString : T_MaxString;
    ActualString : T_MaxString;
    AlreadyReported : BOOL;
    TestInstancePath : T_MaxString;
    SizeOfExpecteds : DINT;
    SizeOfActuals : DINT;
    ExpectedDWordString : STRING;
    ActualDWordString : STRING;
    ExpectedsIndex : DINT;
    ActualsIndex : DINT;
END_VAR
IF GVL_TcUnit.IgnoreCurrentTest OR GVL_TcUnit.CurrentTestIsFinished THEN
    RETURN;
END_IF

TestInstancePath := AddTestNameToInstancePath(FindTestSuiteInstancePath());

SizeOfExpecteds := ABS(UPPER_BOUND(Expecteds, 1) - LOWER_BOUND(Expecteds, 1)) + 1;
SizeOfActuals := ABS(UPPER_BOUND(Actuals, 1) - LOWER_BOUND(Actuals, 1)) + 1;

IF SizeOfExpecteds <> SizeOfActuals THEN
    Equals := FALSE;
    SizeEquals := FALSE;
ELSE
    (* Even though we know that both arrays are equal in size, the two arrays can start at two completely different
       indexes, which needs to be taken into account for. *)
    ExpectedsIndex := LOWER_BOUND(Expecteds, 1); // The start position for the expecteds
    ActualsIndex := LOWER_BOUND(Actuals, 1); // The start position for the actuals
    FOR Index := 1 TO SizeOfExpecteds BY 1 DO
        IF Expecteds[ExpectedsIndex] <> Actuals[ActualsIndex] THEN
            Equals := FALSE;
            EXIT;
        END_IF
        ExpectedsIndex := ExpectedsIndex + 1;
        ActualsIndex := ActualsIndex + 1;
    END_FOR
END_IF

AssertArrayResults.ReportResult(ExpectedsSize := DINT_TO_UDINT(SizeOfExpecteds),
                                ExpectedsTypeClass := IBaseLibrary.TypeClass.TYPE_DWORD,
                                ActualsSize := DINT_TO_UDINT(SizeOfActuals),
                                ActualsTypeClass := IBaseLibrary.TypeClass.TYPE_DWORD,
                                Message := Message,
                                TestInstancePath := TestInstancePath,
                                AlreadyReported => AlreadyReported);

IF NOT AlreadyReported AND NOT Equals THEN
    SetTestFailed(AssertionType := E_AssertionType.Type_Array_DWORD,
                  AssertionMessage := Message);
    
    IF NOT SizeEquals THEN
        Message := CONCAT(STR1 := Message, STR2 := ', size of arrays not matching.');
        ExpectedString := 'SIZE = ';
        ExpectedString := CONCAT(STR1 := ExpectedString, STR2 := DINT_TO_STRING(SizeOfExpecteds));
        ActualString := 'SIZE = ';
        ActualString := CONCAT(STR1 := ActualString, STR2 := DINT_TO_STRING(SizeOfActuals));
    ELSE
        ExpectedDWordString := CONCAT(STR1 := '0x',
                                                   STR2 := DWORD_TO_HEXSTR(in := Expecteds[ExpectedsIndex],
                                                                                         iPrecision := 8,
                                                                                         bLoCase := FALSE));
        ExpectedString := 'ARRAY[';
        ExpectedString := CONCAT(STR1 := ExpectedString, STR2 := DINT_TO_STRING(ExpectedsIndex));
        ExpectedString := CONCAT(STR1 := ExpectedString, STR2 := '] = ');
        ExpectedString := CONCAT(STR1 := ExpectedString, STR2 := ExpectedDWordString);

        ActualDWordString := CONCAT(STR1 := '0x',
                                                 STR2 := DWORD_TO_HEXSTR(in := Actuals[ActualsIndex],
                                                                                       iPrecision := 8,
                                                                                       bLoCase := FALSE));
        ActualString := 'ARRAY[';
        ActualString := CONCAT(STR1 := ActualString, STR2 := DINT_TO_STRING(ActualsIndex));
        ActualString := CONCAT(STR1 := ActualString, STR2 := '] = ');
        ActualString := CONCAT(STR1 := ActualString, STR2 := ActualDWordString);
    END_IF

    AssertMessageFormatter.LogAssertFailure(Expected := ExpectedString,
                                            Actual := ActualString,
                                            Message := Message,
                                            TestInstancePath := TestInstancePath);
END_IF
END_METHOD

// Asserts that two INT arrays are equal. If they are not, an assertion error is created.
METHOD PUBLIC AssertArrayEquals_INT
VAR_IN_OUT
    Expecteds : ARRAY[*] OF INT; // INT array with expected values
    Actuals : ARRAY[*] OF INT; // INT array with actual values
END_VAR
VAR_INPUT
    Message : T_MaxString; // The identifying message for the assertion error
END_VAR
VAR
    Equals : BOOL := TRUE;
    SizeEquals : BOOL := TRUE;
    Index : DINT;
    ExpectedString : T_MaxString;
    ActualString : T_MaxString;
    AlreadyReported : BOOL;
    TestInstancePath : T_MaxString;
    SizeOfExpecteds : DINT;
    SizeOfActuals : DINT;
    ExpectedsIndex : DINT;
    ActualsIndex : DINT;
END_VAR
IF GVL_TcUnit.IgnoreCurrentTest OR GVL_TcUnit.CurrentTestIsFinished THEN
    RETURN;
END_IF

TestInstancePath := AddTestNameToInstancePath(FindTestSuiteInstancePath());

SizeOfExpecteds := ABS(UPPER_BOUND(Expecteds, 1) - LOWER_BOUND(Expecteds, 1)) + 1;
SizeOfActuals := ABS(UPPER_BOUND(Actuals, 1) - LOWER_BOUND(Actuals, 1)) + 1;

IF SizeOfExpecteds <> SizeOfActuals THEN
    Equals := FALSE;
    SizeEquals := FALSE;
ELSE
    (* Even though we know that both arrays are equal in size, the two arrays can start at two completely different
       indexes, which needs to be taken into account for. *)
    ExpectedsIndex := LOWER_BOUND(Expecteds, 1); // The start position for the expecteds
    ActualsIndex := LOWER_BOUND(Actuals, 1); // The start position for the actuals
    FOR Index := 1 TO SizeOfExpecteds BY 1 DO
        IF Expecteds[ExpectedsIndex] <> Actuals[ActualsIndex] THEN
            Equals := FALSE;
            EXIT;
        END_IF
        ExpectedsIndex := ExpectedsIndex + 1;
        ActualsIndex := ActualsIndex + 1;
    END_FOR
END_IF

AssertArrayResults.ReportResult(ExpectedsSize := DINT_TO_UDINT(SizeOfExpecteds),
                                ExpectedsTypeClass := IBaseLibrary.TypeClass.TYPE_INT,
                                ActualsSize := DINT_TO_UDINT(SizeOfActuals),
                                ActualsTypeClass := IBaseLibrary.TypeClass.TYPE_INT,
                                Message := Message,
                                TestInstancePath := TestInstancePath,
                                AlreadyReported => AlreadyReported);

IF NOT AlreadyReported AND NOT Equals THEN
    SetTestFailed(AssertionType := E_AssertionType.Type_Array_INT,
                  AssertionMessage := Message);

    IF NOT SizeEquals THEN
        Message := CONCAT(STR1 := Message, STR2 := ', size of arrays not matching.');
        ExpectedString := 'SIZE = ';
        ExpectedString := CONCAT(STR1 := ExpectedString, STR2 := DINT_TO_STRING(SizeOfExpecteds));
        ActualString := 'SIZE = ';
        ActualString := CONCAT(STR1 := ActualString, STR2 := DINT_TO_STRING(SizeOfActuals));
    ELSE
        ExpectedString := 'ARRAY[';
        ExpectedString := CONCAT(STR1 := ExpectedString, STR2 := DINT_TO_STRING(ExpectedsIndex));
        ExpectedString := CONCAT(STR1 := ExpectedString, STR2 := '] = ');
        ExpectedString := CONCAT(STR1 := ExpectedString, STR2 := INT_TO_STRING(Expecteds[ExpectedsIndex]));

        ActualString := 'ARRAY[';
        ActualString := CONCAT(STR1 := ActualString, STR2 := DINT_TO_STRING(ActualsIndex));
        ActualString := CONCAT(STR1 := ActualString, STR2 := '] = ');
        ActualString := CONCAT(STR1 := ActualString, STR2 := INT_TO_STRING(Actuals[ActualsIndex]));
    END_IF

